IF im.v3_Avom.onStatus=statusDualInput.status_on THEN
	narabotka_izm:=DT_TO_UDINT( timer.CDT);
	timer.EN:=TRUE;
ELSE
	timer.EN:=FALSE;
END_IF
narabotka_hour (clk:=(narabotka_izm >=3600));
IF	narabotka_hour.Q THEN
	narabotka:=narabotka+1;
	timer.EN:=FALSE;
	narabotka_izm:=0;
END_IF
timer();

saveTimer(IN:=true);
IF saveTimer.Q THEN
	SaveToFile();
	saveTimer(IN:=FALSE);
END_IF*)

METHOD PROTECTED readPersistent
VAR_INPUT
END_VAR

narabotka:=STRING_TO_UDINT(readValue());
narabotka_izm:=STRING_TO_UDINT(readValue());
END_METHOD

METHOD PROTECTED writePersistent
VAR_INPUT
END_VAR

writeValue(value:= UDINT_TO_STRING(narabotka),'Наработка');
writeValue(value:= UDINT_TO_STRING(narabotka_izm),'Наработка_izm');
END_METHOD

END_FUNCTION_BLOCK

// K2/std12k5/Natabotka/Avom3
	{attribute 'symbol' := 'none'}
FUNCTION_BLOCK Avom3 EXTENDS Vent
VAR_INPUT
END_VAR
VAR_OUTPUT
		{attribute 'symbol' := 'read'}
	narabotka:UDINT;
	narabotka_:ExtNarabotka (table:=ADR (objectTable)):=(saveInterval:=T#1H);
END_VAR
VAR
	(*timer:RTC;	
	saveTimer:TON:=(PT:=T#600S);
	Narabotka_hour:R_TRIG;
	AvomStartted:R_TRIG;
	narabotka_Izm:UDINT;*)
END_VAR

SUPER^();
narabotka_.started:=onstatus=statusDualInput.STATUS_ON;
narabotka:=(narabotka_.narabotka/3600);
(*

AvomStartted(CLK:=im.v3_Avom.onStatus=statusDualInput.status_on);

	timer.PDT:=UDINT_TO_DT(narabotka_izm);

IF im.v3_Avom.onStatus=statusDualInput.status_on THEN
	narabotka_izm:=DT_TO_UDINT( timer.CDT);
	timer.EN:=TRUE;
ELSE
	timer.EN:=FALSE;
END_IF
narabotka_hour (clk:=(narabotka_izm >=3600));
IF	narabotka_hour.Q THEN
	narabotka:=narabotka+1;
	timer.EN:=FALSE;
	narabotka_izm:=0;
END_IF
timer();

saveTimer(IN:=true);
IF saveTimer.Q THEN
	SaveToFile();
	saveTimer(IN:=FALSE);
END_IF*)

METHOD PROTECTED readPersistent
VAR_INPUT
END_VAR

narabotka:=STRING_TO_UDINT(readValue());
narabotka_izm:=STRING_TO_UDINT(readValue());
END_METHOD

METHOD PROTECTED writePersistent
VAR_INPUT
END_VAR

writeValue(value:= UDINT_TO_STRING(narabotka),'Наработка');
writeValue(value:= UDINT_TO_STRING(narabotka_izm),'Наработка_izm');
END_METHOD

END_FUNCTION_BLOCK

// K1/std12k5/Narabotka/Avom4
	{attribute 'symbol' := 'none'}
FUNCTION_BLOCK Avom4 EXTENDS Vent
VAR_INPUT
END_VAR
VAR_OUTPUT
		{attribute 'symbol' := 'read'}
	narabotka:UDINT;
	narabotka_:ExtNarabotka (table:=ADR (objectTable)):=(saveInterval:=T#1H);
END_VAR
VAR
	(*timer:RTC;	
	saveTimer:TON:=(PT:=T#600S);
	Narabotka_hour:R_TRIG;
	AvomStartted:R_TRIG;
	narabotka_Izm:UDINT;*)
END_VAR

SUPER^();
narabotka_.started:=onstatus=statusDualInput.STATUS_ON;
narabotka:=(narabotka_.narabotka/3600);
(*
AvomStartted(CLK:=im.v4_Avom.onStatus=statusDualInput.status_on);

	timer.PDT:=UDINT_TO_DT(narabotka_izm);

IF im.v4_Avom.onStatus=statusDualInput.status_on THEN
	narabotka_izm:=DT_TO_UDINT( timer.CDT);
	timer.EN:=TRUE;
ELSE
	timer.EN:=FALSE;
END_IF
narabotka_hour (clk:=(narabotka_izm >=3600));
IF	narabotka_hour.Q THEN
	narabotka:=narabotka+1;
	timer.EN:=FALSE;
	narabotka_izm:=0;
END_IF
timer();

saveTimer(IN:=true);
IF saveTimer.Q THEN
	SaveToFile();
	saveTimer(IN:=FALSE);
END_IF*)

METHOD PROTECTED readPersistent
VAR_INPUT
END_VAR

narabotka:=STRING_TO_UDINT(readValue());
narabotka_izm:=STRING_TO_UDINT(readValue());
END_METHOD

METHOD PROTECTED writePersistent
VAR_INPUT
END_VAR

writeValue(value:= UDINT_TO_STRING(narabotka),'Наработка');
writeValue(value:= UDINT_TO_STRING(narabotka_izm),'Наработка_izm');
END_METHOD

END_FUNCTION_BLOCK

// K2/std12k5/Natabotka/Avom4
	{attribute 'symbol' := 'none'}
FUNCTION_BLOCK Avom4 EXTENDS Vent
VAR_INPUT
END_VAR
VAR_OUTPUT
		{attribute 'symbol' := 'read'}
	narabotka:UDINT;
	narabotka_:ExtNarabotka (table:=ADR (objectTable)):=(saveInterval:=T#1H);
END_VAR
VAR
(*	timer:RTC;	
	saveTimer:TON:=(PT:=T#600S);
	Narabotka_hour:R_TRIG;
	AvomStartted:R_TRIG;
	narabotka_Izm:UDINT;*)
END_VAR

SUPER^();
narabotka_.started:=onstatus=statusDualInput.STATUS_ON;
narabotka:=(narabotka_.narabotka/3600);

(*
AvomStartted(CLK:=im.v4_Avom.onStatus=statusDualInput.status_on);

	timer.PDT:=UDINT_TO_DT(narabotka_izm);

IF im.v4_Avom.onStatus=statusDualInput.status_on THEN
	narabotka_izm:=DT_TO_UDINT( timer.CDT);
	timer.EN:=TRUE;
ELSE
	timer.EN:=FALSE;
END_IF
narabotka_hour (clk:=(narabotka_izm >=3600));
IF	narabotka_hour.Q THEN
	narabotka:=narabotka+1;
	timer.EN:=FALSE;
	narabotka_izm:=0;
END_IF
timer();

saveTimer(IN:=true);
IF saveTimer.Q THEN
	SaveToFile();
	saveTimer(IN:=FALSE);
END_IF*)

METHOD PROTECTED readPersistent
VAR_INPUT
END_VAR

narabotka:=STRING_TO_UDINT(readValue());
narabotka_izm:=STRING_TO_UDINT(readValue());
END_METHOD

METHOD PROTECTED writePersistent
VAR_INPUT
END_VAR

writeValue(value:= UDINT_TO_STRING(narabotka),'Наработка');
writeValue(value:= UDINT_TO_STRING(narabotka_izm),'Наработка_izm');
END_METHOD

END_FUNCTION_BLOCK

// K1/std12k5/Ystavki/Delta_Vykl_AVOM1
	{attribute 'symbol' := 'none'}
FUNCTION_BLOCK Delta_Vykl_AVOM1 EXTENDS Baseobject
VAR_INPUT
	{attribute 'symbol' := 'readwright'}
	Yst_izm:UINT;
END_VAR
VAR_OUTPUT
	{attribute 'symbol' := 'read'}
	Yst_T1:UINT;
	
END_VAR
VAR
	Yst_Izm_trig:R_TRIG;
	Yst_First_izm:R_TRIG;
	flag:bool;
END_VAR

SUPER^();
Yst_Izm_trig(clk:=((Yst_izm <> Yst_T1) AND (Yst_izm >0) AND (Yst_izm <= 10)));
IF 	Yst_Izm_trig.Q THEN
	Yst_T1 := Yst_izm;
	SaveToFile();
END_IF	
Yst_First_izm(clk:=((Yst_izm = 0) AND (Yst_T1 = 0) AND flag));
IF	(Yst_izm = 0) AND (Yst_T1 = 0) AND flag THEN
	Yst_T1 := 1;
	Yst_izm := Yst_T1;
	SaveToFile();
END_IF;

flag:=true;

METHOD PROTECTED readPersistent
VAR_INPUT
END_VAR
Yst_izm:=STRING_TO_uint(readValue());
END_METHOD

METHOD PROTECTED writePersistent
VAR_INPUT
END_VAR
writeValue(value:= uint_TO_STRING(Yst_T1),'Наработка');
END_METHOD

END_FUNCTION_BLOCK

// K2/std12k5/Ystavki/Delta_Vykl_AVOM1
	{attribute 'symbol' := 'none'}
FUNCTION_BLOCK Delta_Vykl_AVOM1 EXTENDS Baseobject
VAR_INPUT
	{attribute 'symbol' := 'readwright'}
	Yst_izm:UINT;
END_VAR
VAR_OUTPUT
	{attribute 'symbol' := 'read'}
	Yst_T1:UINT;
	
END_VAR
VAR
	Yst_Izm_trig:R_TRIG;
	Yst_First_izm:R_TRIG;
	flag:bool;
END_VAR

SUPER^();
Yst_Izm_trig(clk:=((Yst_izm <> Yst_T1) AND (Yst_izm >0) AND (Yst_izm <= 10)));
IF 	Yst_Izm_trig.Q THEN
	Yst_T1 := Yst_izm;
	SaveToFile();
END_IF	
Yst_First_izm(clk:=((Yst_izm = 0) AND (Yst_T1 = 0) AND flag));
IF	(Yst_izm = 0) AND (Yst_T1 = 0) AND flag THEN
	Yst_T1 := 1;
	Yst_izm := Yst_T1;
	SaveToFile();
END_IF;

flag:=true;

METHOD PROTECTED readPersistent
VAR_INPUT
END_VAR
Yst_izm:=STRING_TO_uint(readValue());
END_METHOD

METHOD PROTECTED writePersistent
VAR_INPUT
END_VAR
writeValue(value:= uint_TO_STRING(Yst_T1),'Наработка');
END_METHOD

END_FUNCTION_BLOCK

// K1/std12k5/Ystavki/Delta_Vykl_AVOM2
	{attribute 'symbol' := 'none'}
FUNCTION_BLOCK Delta_Vykl_AVOM2 EXTENDS Baseobject
VAR_INPUT
	{attribute 'symbol' := 'readwright'}
	Yst_izm:UINT;
END_VAR
VAR_OUTPUT
	{attribute 'symbol' := 'read'}
	Yst_T2:UINT;
	
END_VAR
VAR
	Yst_Izm_trig:R_TRIG;
	Yst_First_izm:R_TRIG;
	flag:bool;
END_VAR

SUPER^();
Yst_Izm_trig(clk:=((Yst_izm <> Yst_T2) AND (Yst_izm > 0) AND (Yst_izm <=10)));
IF 	Yst_Izm_trig.Q THEN
	Yst_T2 := Yst_izm;
	SaveToFile();
END_IF	
Yst_First_izm(clk:=((Yst_izm = 0) AND (Yst_T2 = 0) AND flag));
IF	Yst_First_izm.Q	THEN
	Yst_T2 := 1;
	Yst_izm := Yst_T2;
	SaveToFile();
END_IF;
flag:=TRUE;

METHOD PROTECTED readPersistent
VAR_INPUT
END_VAR
Yst_izm:=STRING_TO_uint(readValue());
END_METHOD

METHOD PROTECTED writePersistent
VAR_INPUT
END_VAR
writeValue(value:= uint_TO_STRING(Yst_T2),'Наработка');
END_METHOD

END_FUNCTION_BLOCK

// K2/std12k5/Ystavki/Delta_Vykl_AVOM2
	{attribute 'symbol' := 'none'}
FUNCTION_BLOCK Delta_Vykl_AVOM2 EXTENDS Baseobject
VAR_INPUT
	{attribute 'symbol' := 'readwright'}
	Yst_izm:UINT;
END_VAR
VAR_OUTPUT
	{attribute 'symbol' := 'read'}
	Yst_T2:UINT;
	
END_VAR
VAR
	Yst_Izm_trig:R_TRIG;
	Yst_First_izm:R_TRIG;
	flag:bool;
END_VAR

SUPER^();
Yst_Izm_trig(clk:=((Yst_izm <> Yst_T2) AND (Yst_izm > 0) AND (Yst_izm <=10)));
IF 	Yst_Izm_trig.Q THEN
	Yst_T2 := Yst_izm;
	SaveToFile();
END_IF	
Yst_First_izm(clk:=((Yst_izm = 0) AND (Yst_T2 = 0) AND flag));
IF	Yst_First_izm.Q	THEN
	Yst_T2 := 1;
	Yst_izm := Yst_T2;
	SaveToFile();
END_IF;
flag:=TRUE;

METHOD PROTECTED readPersistent
VAR_INPUT
END_VAR
Yst_izm:=STRING_TO_uint(readValue());
END_METHOD

METHOD PROTECTED writePersistent
VAR_INPUT
END_VAR
writeValue(value:= uint_TO_STRING(Yst_T2),'Наработка');
END_METHOD

END_FUNCTION_BLOCK

// K1/std12k5/Ystavki/Delta_Vykl_AVOM3
	{attribute 'symbol' := 'none'}
FUNCTION_BLOCK Delta_Vykl_AVOM3 EXTENDS Baseobject
VAR_INPUT
	{attribute 'symbol' := 'readwright'}
	Yst_izm:UINT;
END_VAR
VAR_OUTPUT
	{attribute 'symbol' := 'read'}
	Yst_T3:UINT;
	
END_VAR
VAR
	flag:BOOL;
	Yst_Izm_trig:R_TRIG;
	Yst_First_izm:R_TRIG;
END_VAR

SUPER^();
Yst_Izm_trig(clk:=((Yst_izm <> Yst_T3) AND (Yst_izm >0) AND (Yst_izm <= 10)));
IF 	Yst_Izm_trig.Q THEN
	Yst_T3 := Yst_izm;
	SaveToFile();
END_IF	
Yst_First_izm(clk:=((Yst_izm = 0) AND (Yst_T3 = 0) AND flag));
IF	Yst_First_izm.Q THEN
	Yst_T3 := 1;
	Yst_izm := Yst_T3;
	SaveToFile();
END_IF;
flag:=true;

METHOD PROTECTED readPersistent
VAR_INPUT
END_VAR

Yst_izm:=STRING_TO_uint(readValue());
END_METHOD

METHOD PROTECTED writePersistent
VAR_INPUT
END_VAR

writeValue(value:= uint_TO_STRING(Yst_T3),'Наработка');
END_METHOD

END_FUNCTION_BLOCK

// K2/std12k5/Ystavki/Delta_Vykl_AVOM3
	{attribute 'symbol' := 'none'}
FUNCTION_BLOCK Delta_Vykl_AVOM3 EXTENDS Baseobject
VAR_INPUT
	{attribute 'symbol' := 'readwright'}
	Yst_izm:UINT;
END_VAR
VAR_OUTPUT
	{attribute 'symbol' := 'read'}
	Yst_T3:UINT;
	
END_VAR
VAR
	flag:BOOL;
	Yst_Izm_trig:R_TRIG;
	Yst_First_izm:R_TRIG;
END_VAR

SUPER^();
Yst_Izm_trig(clk:=((Yst_izm <> Yst_T3) AND (Yst_izm >0) AND (Yst_izm <= 10)));
IF 	Yst_Izm_trig.Q THEN
	Yst_T3 := Yst_izm;
	SaveToFile();
END_IF	
Yst_First_izm(clk:=((Yst_izm = 0) AND (Yst_T3 = 0) AND flag));
IF	Yst_First_izm.Q THEN
	Yst_T3 := 1;
	Yst_izm := Yst_T3;
	SaveToFile();
END_IF;
flag:=true;

METHOD PROTECTED readPersistent
VAR_INPUT
END_VAR

Yst_izm:=STRING_TO_uint(readValue());
END_METHOD

METHOD PROTECTED writePersistent
VAR_INPUT
END_VAR

writeValue(value:= uint_TO_STRING(Yst_T3),'Наработка');
END_METHOD

END_FUNCTION_BLOCK

// K1/std12k5/Ystavki/Delta_Vykl_AVOM4
	{attribute 'symbol' := 'none'}
FUNCTION_BLOCK Delta_Vykl_AVOM4 EXTENDS Baseobject
VAR_INPUT
	{attribute 'symbol' := 'readwright'}
	Yst_izm:UINT;
END_VAR
VAR_OUTPUT
	{attribute 'symbol' := 'read'}
	Yst_T4:UINT;
	
END_VAR
VAR
	flag:BOOL;
	Yst_Izm_trig:R_TRIG;
	Yst_First_izm:R_TRIG;
END_VAR

SUPER^();
Yst_Izm_trig(clk:=((Yst_izm <> Yst_T4) AND (Yst_izm > 0) AND (Yst_izm <= 10)));
IF 	Yst_Izm_trig.Q THEN
	Yst_T4 := Yst_izm;
	SaveToFile();
END_IF	
Yst_First_izm(clk:=((Yst_izm = 0) AND (Yst_T4 = 0) AND flag));
IF	Yst_First_izm.Q THEN
	Yst_T4 := 1;
	Yst_izm := Yst_T4;
	SaveToFile();
END_IF;

flag:=TRUE;

METHOD PROTECTED readPersistent
VAR_INPUT
END_VAR

Yst_izm:=STRING_TO_uint(readValue());
END_METHOD

METHOD PROTECTED writePersistent
VAR_INPUT
END_VAR

writeValue(value:= uint_TO_STRING(Yst_T4),'Наработка');
END_METHOD

END_FUNCTION_BLOCK

// K2/std12k5/Ystavki/Delta_Vykl_AVOM4
	{attribute 'symbol' := 'none'}
FUNCTION_BLOCK Delta_Vykl_AVOM4 EXTENDS Baseobject
VAR_INPUT
	{attribute 'symbol' := 'readwright'}
	Yst_izm:UINT;
END_VAR
VAR_OUTPUT
	{attribute 'symbol' := 'read'}
	Yst_T4:UINT;
	
END_VAR
VAR
	flag:BOOL;
	Yst_Izm_trig:R_TRIG;
	Yst_First_izm:R_TRIG;
END_VAR

SUPER^();
Yst_Izm_trig(clk:=((Yst_izm <> Yst_T4) AND (Yst_izm > 0) AND (Yst_izm <= 10)));
IF 	Yst_Izm_trig.Q THEN
	Yst_T4 := Yst_izm;
	SaveToFile();
END_IF	
Yst_First_izm(clk:=((Yst_izm = 0) AND (Yst_T4 = 0) AND flag));
IF	Yst_First_izm.Q THEN
	Yst_T4 := 1;
	Yst_izm := Yst_T4;
	SaveToFile();
END_IF;

flag:=TRUE;

METHOD PROTECTED readPersistent
VAR_INPUT
END_VAR

Yst_izm:=STRING_TO_uint(readValue());
END_METHOD

METHOD PROTECTED writePersistent
VAR_INPUT
END_VAR

writeValue(value:= uint_TO_STRING(Yst_T4),'Наработка');
END_METHOD

END_FUNCTION_BLOCK

// K1/std12k5/Narabotka/EO
	{attribute 'symbol' := 'none'}
FUNCTION_BLOCK EO EXTENDS BaseIM
VAR_INPUT
END_VAR
VAR_OUTPUT
	
		{attribute 'symbol' := 'read'}
	narabotka:UDINT;
END_VAR
VAR
	Work_End:F_TRIG;
	flag:bool;
	AvomStartted:R_TRIG;
END_VAR

SUPER^();
Work_END (CLK:=(algmanager.mode=modegpa.MODE_WORK_K OR algmanager.mode=modegpa.MODE_WORK_M));
IF Work_END.Q THEN
	flag:=TRUE;
END_IF
AvomStartted(CLK:=(algmanager.mode=modegpa.MODE_EO) AND flag);
IF AvomStartted.Q THEN
	narabotka:= narabotka + 1;
	SaveToFile();
	flag:=false;
END_IF

METHOD PROTECTED readPersistent
VAR_INPUT
END_VAR

narabotka:=STRING_TO_UDINT(readValue());
END_METHOD

METHOD PROTECTED writePersistent
VAR_INPUT
END_VAR

writeValue(value:= UDINT_TO_STRING(narabotka),'Наработка');
END_METHOD

END_FUNCTION_BLOCK

// K2/std12k5/Natabotka/EO
	{attribute 'symbol' := 'none'}
FUNCTION_BLOCK EO EXTENDS BaseIM
VAR_INPUT
END_VAR
VAR_OUTPUT
	
		{attribute 'symbol' := 'read'}
	narabotka:UDINT;
END_VAR
VAR
	Work_End:F_TRIG;
	flag:bool;
	AvomStartted:R_TRIG;
END_VAR

SUPER^();
Work_END (CLK:=(algmanager.mode=modegpa.MODE_WORK_K OR algmanager.mode=modegpa.MODE_WORK_M));
IF Work_END.Q THEN
	flag:=TRUE;
END_IF
AvomStartted(CLK:=(algmanager.mode=modegpa.MODE_EO) AND flag);
IF AvomStartted.Q THEN
	narabotka:= narabotka + 1;
	SaveToFile();
	flag:=false;
END_IF

METHOD PROTECTED readPersistent
VAR_INPUT
END_VAR

narabotka:=STRING_TO_UDINT(readValue());
END_METHOD

METHOD PROTECTED writePersistent
VAR_INPUT
END_VAR

writeValue(value:= UDINT_TO_STRING(narabotka),'Наработка');
END_METHOD

END_FUNCTION_BLOCK

// K1/std12k5/Narabotka/nu1
	{attribute 'symbol' := 'none'}
FUNCTION_BLOCK nu1 EXTENDS nasos
VAR_INPUT
END_VAR
VAR_OUTPUT
	
		{attribute 'symbol' := 'read'}
	narabotka:UDINT;
	narabotka_:ExtNarabotka (table:=ADR (objectTable)):=(saveInterval:=T#1H);
END_VAR
VAR
	(*	timer:RTC;	
	saveTimer:TON:=(PT:=T#600S);
	Narabotka_hour:R_TRIG;
	AvomStartted:R_TRIG;
	narabotka_Izm:UDINT;*)
END_VAR

SUPER^();
narabotka_.started:=im.nu.nu1.onStatus=statusDualInput.STATUS_ON;
narabotka:=(narabotka_.narabotka/3600);
(*
AvomStartted(CLK:=im.nu.nu1.onStatus=statusDualInput.status_on);

	timer.PDT:=UDINT_TO_DT(narabotka_izm);

IF im.nu.nu1.onStatus=statusDualInput.status_on THEN
	narabotka_izm:=DT_TO_UDINT( timer.CDT);
	timer.EN:=TRUE;
ELSE
	timer.EN:=FALSE;
END_IF
narabotka_hour (clk:=(narabotka_izm >=3600));
IF	narabotka_hour.Q THEN
	narabotka:=narabotka+1;
	timer.EN:=FALSE;
	narabotka_izm:=0;
END_IF
timer();

saveTimer(IN:=true);
IF saveTimer.Q THEN
	SaveToFile();
	saveTimer(IN:=FALSE);
END_IF*)

METHOD PROTECTED readPersistent
VAR_INPUT
END_VAR

narabotka:=STRING_TO_UDINT(readValue());
narabotka_izm:=STRING_TO_UDINT(readValue());
END_METHOD

METHOD PROTECTED writePersistent
VAR_INPUT
END_VAR

writeValue(value:= UDINT_TO_STRING(narabotka),'Наработка');
writeValue(value:= UDINT_TO_STRING(narabotka_izm),'Наработка_izm');
END_METHOD

END_FUNCTION_BLOCK

// K2/std12k5/Natabotka/nu1
	{attribute 'symbol' := 'none'}
FUNCTION_BLOCK nu1 EXTENDS nasos
VAR_INPUT
END_VAR
VAR_OUTPUT
	
		{attribute 'symbol' := 'read'}
	narabotka:UDINT;
	narabotka_:ExtNarabotka (table:=ADR (objectTable)):=(saveInterval:=T#1H);
END_VAR
VAR
	(*	timer:RTC;	
	saveTimer:TON:=(PT:=T#600S);
	Narabotka_hour:R_TRIG;
	AvomStartted:R_TRIG;
	narabotka_Izm:UDINT;*)
END_VAR

SUPER^();
narabotka_.started:=im.nu.nu1.onStatus=statusDualInput.STATUS_ON;
narabotka:=(narabotka_.narabotka/3600);
(*
AvomStartted(CLK:=im.nu.nu1.onStatus=statusDualInput.status_on);

	timer.PDT:=UDINT_TO_DT(narabotka_izm);

IF im.nu.nu1.onStatus=statusDualInput.status_on THEN
	narabotka_izm:=DT_TO_UDINT( timer.CDT);
	timer.EN:=TRUE;
ELSE
	timer.EN:=FALSE;
END_IF
narabotka_hour (clk:=(narabotka_izm >=3600));
IF	narabotka_hour.Q THEN
	narabotka:=narabotka+1;
	timer.EN:=FALSE;
	narabotka_izm:=0;
END_IF
timer();

saveTimer(IN:=true);
IF saveTimer.Q THEN
	SaveToFile();
	saveTimer(IN:=FALSE);
END_IF*)

METHOD PROTECTED readPersistent
VAR_INPUT
END_VAR

narabotka:=STRING_TO_UDINT(readValue());
narabotka_izm:=STRING_TO_UDINT(readValue());
END_METHOD

METHOD PROTECTED writePersistent
VAR_INPUT
END_VAR

writeValue(value:= UDINT_TO_STRING(narabotka),'Наработка');
writeValue(value:= UDINT_TO_STRING(narabotka_izm),'Наработка_izm');
END_METHOD

END_FUNCTION_BLOCK

// lowLevel_ecl/im/ventvs/Nasos
	{attribute 'symbol' := 'none'}
FUNCTION_BLOCK Nasos EXTENDS Ventvs
VAR_INPUT
END_VAR
VAR_OUTPUT
END_VAR
VAR
END_VAR

SUPER^();

END_FUNCTION_BLOCK

// K1/std12k5/Narabotka/nu2
	{attribute 'symbol' := 'none'}
FUNCTION_BLOCK nu2 EXTENDS Nasos
VAR_INPUT
END_VAR
VAR_OUTPUT
	
		{attribute 'symbol' := 'read'}
	narabotka:UDINT;
	narabotka_:ExtNarabotka (table:=ADR (objectTable)):=(saveInterval:=T#1H);
END_VAR
VAR
(*	timer:RTC;	
	saveTimer:TON:=(PT:=T#600S);
	Narabotka_hour:R_TRIG;
	AvomStartted:R_TRIG;
	narabotka_Izm:UDINT;*)
END_VAR

SUPER^();
narabotka_.started:=im.nu.nu2.onStatus=statusDualInput.STATUS_ON;
narabotka:=(narabotka_.narabotka/3600);
(*
AvomStartted(CLK:=im.nu.nu2.onStatus=statusDualInput.status_on);

	timer.PDT:=UDINT_TO_DT(narabotka_izm);

IF im.nu.nu2.onStatus=statusDualInput.status_on THEN
	narabotka_izm:=DT_TO_UDINT( timer.CDT);
	timer.EN:=TRUE;
ELSE
	timer.EN:=FALSE;
END_IF
narabotka_hour (clk:=(narabotka_izm >=3600));
IF	narabotka_hour.Q THEN
	narabotka:=narabotka+1;
	timer.EN:=FALSE;
	narabotka_izm:=0;
END_IF
timer();

saveTimer(IN:=true);
IF saveTimer.Q THEN
	SaveToFile();
	saveTimer(IN:=FALSE);
END_IF*)

METHOD PROTECTED readPersistent
VAR_INPUT
END_VAR

narabotka:=STRING_TO_UDINT(readValue());
narabotka_izm:=STRING_TO_UDINT(readValue());
END_METHOD

METHOD PROTECTED writePersistent
VAR_INPUT
END_VAR

writeValue(value:= UDINT_TO_STRING(narabotka),'Наработка');
writeValue(value:= UDINT_TO_STRING(narabotka_izm),'Наработка_izm');
END_METHOD

END_FUNCTION_BLOCK

// K2/std12k5/Natabotka/nu2
	{attribute 'symbol' := 'none'}
FUNCTION_BLOCK nu2 EXTENDS Nasos
VAR_INPUT
END_VAR
VAR_OUTPUT
	
		{attribute 'symbol' := 'read'}
	narabotka:UDINT;
	narabotka_:ExtNarabotka (table:=ADR (objectTable)):=(saveInterval:=T#1H);
END_VAR
VAR
(*	timer:RTC;	
	saveTimer:TON:=(PT:=T#600S);
	Narabotka_hour:R_TRIG;
	AvomStartted:R_TRIG;
	narabotka_Izm:UDINT;*)
END_VAR

SUPER^();
narabotka_.started:=im.nu.nu2.onStatus=statusDualInput.STATUS_ON;
narabotka:=(narabotka_.narabotka/3600);
(*
AvomStartted(CLK:=im.nu.nu2.onStatus=statusDualInput.status_on);

	timer.PDT:=UDINT_TO_DT(narabotka_izm);

IF im.nu.nu2.onStatus=statusDualInput.status_on THEN
	narabotka_izm:=DT_TO_UDINT( timer.CDT);
	timer.EN:=TRUE;
ELSE
	timer.EN:=FALSE;
END_IF
narabotka_hour (clk:=(narabotka_izm >=3600));
IF	narabotka_hour.Q THEN
	narabotka:=narabotka+1;
	timer.EN:=FALSE;
	narabotka_izm:=0;
END_IF
timer();

saveTimer(IN:=true);
IF saveTimer.Q THEN
	SaveToFile();
	saveTimer(IN:=FALSE);
END_IF*)

METHOD PROTECTED readPersistent
VAR_INPUT
END_VAR

narabotka:=STRING_TO_UDINT(readValue());
narabotka_izm:=STRING_TO_UDINT(readValue());
END_METHOD

METHOD PROTECTED writePersistent
VAR_INPUT
END_VAR

writeValue(value:= UDINT_TO_STRING(narabotka),'Наработка');
writeValue(value:= UDINT_TO_STRING(narabotka_izm),'Наработка_izm');
END_METHOD

END_FUNCTION_BLOCK

// K1/std12k5/Narabotka/pns_
	{attribute 'symbol' := 'none'}
FUNCTION_BLOCK pns_ EXTENDS nasos
VAR_INPUT
END_VAR
VAR_OUTPUT
	
		{attribute 'symbol' := 'read'}
	narabotka:UDINT;
	narabotka_:ExtNarabotka (table:=ADR (objectTable)):=(saveInterval:=T#1H);
END_VAR
VAR
(*	timer:RTC;	
	saveTimer:TON:=(PT:=T#600S);
	Narabotka_hour:R_TRIG;
	AvomStartted:R_TRIG;
	narabotka_Izm:UDINT;*)
END_VAR

SUPER^();
narabotka_.started:=onStatus=statusDualInput.STATUS_ON;
narabotka:=(narabotka_.narabotka/3600);
(*
AvomStartted(CLK:=im.PNS.onStatus=statusDualInput.status_on);

	timer.PDT:=UDINT_TO_DT(narabotka_izm);

IF im.PNS.onStatus=statusDualInput.status_on THEN
	narabotka_izm:=DT_TO_UDINT( timer.CDT);
	timer.EN:=TRUE;
ELSE
	timer.EN:=FALSE;
END_IF
narabotka_hour (clk:=(narabotka_izm >=3600));
IF	narabotka_hour.Q THEN
	narabotka:=narabotka+1;
	timer.EN:=FALSE;
	narabotka_izm:=0;
END_IF
timer();

saveTimer(IN:=true);
IF saveTimer.Q THEN
	SaveToFile();
	saveTimer(IN:=FALSE);
END_IF*)

METHOD PROTECTED readPersistent
VAR_INPUT
END_VAR

narabotka:=STRING_TO_UDINT(readValue());
narabotka_izm:=STRING_TO_UDINT(readValue());
END_METHOD

METHOD PROTECTED writePersistent
VAR_INPUT
END_VAR

writeValue(value:= UDINT_TO_STRING(narabotka),'Наработка');
writeValue(value:= UDINT_TO_STRING(narabotka_izm),'Наработка_izm');
END_METHOD

END_FUNCTION_BLOCK

// K2/std12k5/Natabotka/pns_
	{attribute 'symbol' := 'none'}
FUNCTION_BLOCK pns_ EXTENDS nasos
VAR_INPUT
END_VAR
VAR_OUTPUT
	
		{attribute 'symbol' := 'read'}
	narabotka:UDINT;
		narabotka_:ExtNarabotka (table:=ADR (objectTable)):=(saveInterval:=T#1H);
END_VAR
VAR
	(*timer:RTC;	
	saveTimer:TON:=(PT:=T#600S);
	Narabotka_hour:R_TRIG;
	AvomStartted:R_TRIG;
	narabotka_Izm:UDINT;*)
END_VAR

SUPER^();
narabotka_.started:=onStatus=statusDualInput.STATUS_ON;
narabotka:=(narabotka_.narabotka/3600);
(*
AvomStartted(CLK:=im.PNS.onStatus=statusDualInput.status_on);

	timer.PDT:=UDINT_TO_DT(narabotka_izm);

IF im.PNS.onStatus=statusDualInput.status_on THEN
	narabotka_izm:=DT_TO_UDINT( timer.CDT);
	timer.EN:=TRUE;
ELSE
	timer.EN:=FALSE;
END_IF
narabotka_hour (clk:=(narabotka_izm >=3600));
IF	narabotka_hour.Q THEN
	narabotka:=narabotka+1;
	timer.EN:=FALSE;
	narabotka_izm:=0;
END_IF
timer();

saveTimer(IN:=true);
IF saveTimer.Q THEN
	SaveToFile();
	saveTimer(IN:=FALSE);
END_IF*)

METHOD PROTECTED readPersistent
VAR_INPUT
END_VAR

narabotka:=STRING_TO_UDINT(readValue());
narabotka_izm:=STRING_TO_UDINT(readValue());
END_METHOD

METHOD PROTECTED writePersistent
VAR_INPUT
END_VAR

writeValue(value:= UDINT_TO_STRING(narabotka),'Наработка');
writeValue(value:= UDINT_TO_STRING(narabotka_izm),'Наработка_izm');
END_METHOD

END_FUNCTION_BLOCK

// K1/std12k5/Narabotka/Pusk
	{attribute 'symbol' := 'none'}
FUNCTION_BLOCK Pusk EXTENDS BaseIM
VAR_INPUT
END_VAR
VAR_OUTPUT
	
		{attribute 'symbol' := 'read'}
	narabotka:UDINT;
END_VAR
VAR
	
	
	AvomStartted:R_TRIG;
END_VAR

SUPER^();

AvomStartted(CLK:=(algmanager.mode=modegpa.MODE_WORK_K) OR (algmanager.mode=modegpa.MODE_WORK_M));
IF AvomStartted.Q THEN
	narabotka:= narabotka + 1;
	SaveToFile();
END_IF

METHOD PROTECTED readPersistent
VAR_INPUT
END_VAR

narabotka:=STRING_TO_UDINT(readValue());
END_METHOD

METHOD PROTECTED writePersistent
VAR_INPUT
END_VAR

writeValue(value:= UDINT_TO_STRING(narabotka),'Наработка');
END_METHOD

END_FUNCTION_BLOCK

// K2/std12k5/Natabotka/Pusk
	{attribute 'symbol' := 'none'}
FUNCTION_BLOCK Pusk EXTENDS BaseIM
VAR_INPUT
END_VAR
VAR_OUTPUT
	
		{attribute 'symbol' := 'read'}
	narabotka:UDINT;
END_VAR
VAR
	
	
	AvomStartted:R_TRIG;
END_VAR

SUPER^();

AvomStartted(CLK:=(algmanager.mode=modegpa.MODE_WORK_K) OR (algmanager.mode=modegpa.MODE_WORK_M));
IF AvomStartted.Q THEN
	narabotka:= narabotka + 1;
	SaveToFile();
END_IF

METHOD PROTECTED readPersistent
VAR_INPUT
END_VAR

narabotka:=STRING_TO_UDINT(readValue());
END_METHOD

METHOD PROTECTED writePersistent
VAR_INPUT
END_VAR

writeValue(value:= UDINT_TO_STRING(narabotka),'Наработка');
END_METHOD

END_FUNCTION_BLOCK

// K1/std12k5/Ystavki/T1_AVOM
	{attribute 'symbol' := 'none'}
FUNCTION_BLOCK T1_AVOM EXTENDS Baseobject
VAR_INPUT
	{attribute 'symbol' := 'readwright'}
	Yst_izm:UINT;
END_VAR
VAR_OUTPUT
	{attribute 'symbol' := 'read'}
	Yst_T1:UINT;
	
END_VAR
VAR
	flag:BOOL;
	Yst_Izm_trig:R_TRIG;
	Yst_First_izm:R_TRIG;
END_VAR

SUPER^();
Yst_Izm_trig(clk:=((Yst_izm <> Yst_T1) 	AND (Yst_izm > 0) AND (Yst_izm < 100) AND (Yst_izm < Ystavki.Yst_AVOM_T2.Yst_T2)));
IF 	Yst_Izm_trig.Q THEN
	Yst_T1 := Yst_izm;
	SaveToFile();
END_IF	
Yst_First_izm(clk:=((Yst_izm = 0) AND (Yst_T1 = 0) AND flag));
IF	Yst_First_izm.Q  THEN
	Yst_T1 := 41;
	Yst_izm := Yst_T1;
	SaveToFile();
END_IF;

flag:=true;

METHOD PROTECTED readPersistent
VAR_INPUT
END_VAR

Yst_izm:=STRING_TO_uint(readValue());
END_METHOD

METHOD PROTECTED writePersistent
VAR_INPUT
END_VAR

writeValue(value:= uint_TO_STRING(Yst_T1),'Наработка');
END_METHOD

END_FUNCTION_BLOCK

// K2/std12k5/Ystavki/T1_AVOM
	{attribute 'symbol' := 'none'}
FUNCTION_BLOCK T1_AVOM EXTENDS Baseobject
VAR_INPUT
	{attribute 'symbol' := 'readwright'}
	Yst_izm:UINT;
END_VAR
VAR_OUTPUT
	{attribute 'symbol' := 'read'}
	Yst_T1:UINT;
	
END_VAR
VAR
	flag:BOOL;
	Yst_Izm_trig:R_TRIG;
	Yst_First_izm:R_TRIG;
END_VAR

SUPER^();
Yst_Izm_trig(clk:=((Yst_izm <> Yst_T1) 	AND (Yst_izm > 0) AND (Yst_izm < 100) AND (Yst_izm < Ystavki.Yst_AVOM_T2.Yst_T2)));
IF 	Yst_Izm_trig.Q THEN
	Yst_T1 := Yst_izm;
	SaveToFile();
END_IF	
Yst_First_izm(clk:=((Yst_izm = 0) AND (Yst_T1 = 0) AND flag));
IF	Yst_First_izm.Q  THEN
	Yst_T1 := 41;
	Yst_izm := Yst_T1;
	SaveToFile();
END_IF;

flag:=true;

METHOD PROTECTED readPersistent
VAR_INPUT
END_VAR

Yst_izm:=STRING_TO_uint(readValue());
END_METHOD

METHOD PROTECTED writePersistent
VAR_INPUT
END_VAR

writeValue(value:= uint_TO_STRING(Yst_T1),'Наработка');
END_METHOD

END_FUNCTION_BLOCK

// K1/std12k5/Ystavki/T2_AVOM
	{attribute 'symbol' := 'none'}
FUNCTION_BLOCK T2_AVOM EXTENDS Baseobject
VAR_INPUT
	{attribute 'symbol' := 'readwright'}
	Yst_izm:UINT;
END_VAR
VAR_OUTPUT
	{attribute 'symbol' := 'read'}
	Yst_T2:UINT;
	
END_VAR
VAR
	flag:BOOL;
	Yst_Izm_trig:R_TRIG;
	Yst_First_izm:R_TRIG;
END_VAR

SUPER^();
Yst_Izm_trig(clk:=((Yst_izm <> Yst_T2) 	AND (Yst_izm >0) AND (Yst_izm < 100) AND (Yst_izm > Ystavki.Yst_AVOM_T1.Yst_T1) AND (Yst_izm < Ystavki.Yst_AVOM_T3.Yst_T3)));
IF 	Yst_Izm_trig.Q THEN
	Yst_T2 := Yst_izm;
	SaveToFile();
END_IF	
Yst_First_izm(clk:=((Yst_izm = 0) AND (Yst_T2 = 0) AND flag ));
IF	Yst_First_izm.Q THEN
	Yst_T2 := 42;
	Yst_izm := Yst_T2;
	SaveToFile();
END_IF;



flag:=TRUE;

METHOD PROTECTED readPersistent
VAR_INPUT
END_VAR

Yst_izm:=STRING_TO_uint(readValue());
END_METHOD

METHOD PROTECTED writePersistent
VAR_INPUT
END_VAR

writeValue(value:= uint_TO_STRING(Yst_T2),'Наработка');
END_METHOD

END_FUNCTION_BLOCK

// K2/std12k5/Ystavki/T2_AVOM
	{attribute 'symbol' := 'none'}
FUNCTION_BLOCK T2_AVOM EXTENDS Baseobject
VAR_INPUT
	{attribute 'symbol' := 'readwright'}
	Yst_izm:UINT;
END_VAR
VAR_OUTPUT
	{attribute 'symbol' := 'read'}
	Yst_T2:UINT;
	
END_VAR
VAR
	flag:BOOL;
	Yst_Izm_trig:R_TRIG;
	Yst_First_izm:R_TRIG;
END_VAR

SUPER^();
Yst_Izm_trig(clk:=((Yst_izm <> Yst_T2) 	AND (Yst_izm >0) AND (Yst_izm < 100) AND (Yst_izm > Ystavki.Yst_AVOM_T1.Yst_T1) AND (Yst_izm < Ystavki.Yst_AVOM_T3.Yst_T3)));
IF 	Yst_Izm_trig.Q THEN
	Yst_T2 := Yst_izm;
	SaveToFile();
END_IF	
Yst_First_izm(clk:=((Yst_izm = 0) AND (Yst_T2 = 0) AND flag ));
IF	Yst_First_izm.Q THEN
	Yst_T2 := 42;
	Yst_izm := Yst_T2;
	SaveToFile();
END_IF;



flag:=TRUE;

METHOD PROTECTED readPersistent
VAR_INPUT
END_VAR

Yst_izm:=STRING_TO_uint(readValue());
END_METHOD

METHOD PROTECTED writePersistent
VAR_INPUT
END_VAR

writeValue(value:= uint_TO_STRING(Yst_T2),'Наработка');
END_METHOD

END_FUNCTION_BLOCK

// K1/std12k5/Ystavki/T3_AVOM
	{attribute 'symbol' := 'none'}
FUNCTION_BLOCK T3_AVOM EXTENDS Baseobject
VAR_INPUT
		
	
{attribute 'symbol' := 'readwright'}
	Yst_izm:UINT;
END_VAR
VAR_OUTPUT
	{attribute 'symbol' := 'read'}
	Yst_T3:UINT;
END_VAR
VAR
	flag:BOOL;
	Yst_Izm_trig:R_TRIG;
	Yst_First_izm:R_TRIG;
END_VAR

SUPER^();
Yst_Izm_trig(clk:=((Yst_izm <> Yst_T3) 	AND (Yst_izm >0) AND (Yst_izm < 100) AND (Yst_izm > ystavki.Yst_AVOM_T2.Yst_T2) AND (Yst_izm < ystavki.Yst_AVOM_T4.Yst_T4)));
IF 	Yst_Izm_trig.Q	THEN
	Yst_T3 := Yst_izm;
	SaveToFile();
END_IF	
Yst_First_izm(clk:=((Yst_izm = 0) AND (Yst_T3 = 0) AND flag));
IF	Yst_First_izm.Q THEN
	Yst_T3 := 43;
	Yst_izm := Yst_T3;
	SaveToFile();
END_IF;


flag:=TRUE;

METHOD PROTECTED readPersistent
VAR_INPUT
END_VAR

Yst_izm:=STRING_TO_uint(readValue());
END_METHOD

METHOD PROTECTED writePersistent
VAR_INPUT
END_VAR

writeValue(value:= uint_TO_STRING(Yst_T3),'Наработка');
END_METHOD

END_FUNCTION_BLOCK

// K2/std12k5/Ystavki/T3_AVOM
	{attribute 'symbol' := 'none'}
FUNCTION_BLOCK T3_AVOM EXTENDS Baseobject
VAR_INPUT
		
	
{attribute 'symbol' := 'readwright'}
	Yst_izm:UINT;
END_VAR
VAR_OUTPUT
	{attribute 'symbol' := 'read'}
	Yst_T3:UINT;
END_VAR
VAR
	flag:BOOL;
	Yst_Izm_trig:R_TRIG;
	Yst_First_izm:R_TRIG;
END_VAR

SUPER^();
Yst_Izm_trig(clk:=((Yst_izm <> Yst_T3) 	AND (Yst_izm >0) AND (Yst_izm < 100) AND (Yst_izm > ystavki.Yst_AVOM_T2.Yst_T2) AND (Yst_izm < ystavki.Yst_AVOM_T4.Yst_T4)));
IF 	Yst_Izm_trig.Q	THEN
	Yst_T3 := Yst_izm;
	SaveToFile();
END_IF	
Yst_First_izm(clk:=((Yst_izm = 0) AND (Yst_T3 = 0) AND flag));
IF	Yst_First_izm.Q THEN
	Yst_T3 := 43;
	Yst_izm := Yst_T3;
	SaveToFile();
END_IF;


flag:=TRUE;

METHOD PROTECTED readPersistent
VAR_INPUT
END_VAR

Yst_izm:=STRING_TO_uint(readValue());
END_METHOD

METHOD PROTECTED writePersistent
VAR_INPUT
END_VAR

writeValue(value:= uint_TO_STRING(Yst_T3),'Наработка');
END_METHOD

END_FUNCTION_BLOCK

// K1/std12k5/Ystavki/T4_AVOM
	{attribute 'symbol' := 'none'}
FUNCTION_BLOCK T4_AVOM EXTENDS Baseobject
VAR_INPUT
	{attribute 'symbol' := 'readwright'}
	Yst_izm:UINT;
END_VAR
VAR_OUTPUT
	{attribute 'symbol' := 'read'}
	Yst_T4:UINT;
	
END_VAR
VAR
	flag:BOOL;
	Yst_Izm_trig:R_TRIG;
	Yst_First_izm:R_TRIG;
END_VAR

SUPER^();
Yst_Izm_trig(clk:=((Yst_izm <> Yst_T4) 	AND (Yst_izm >0) AND (Yst_izm < 100) AND (Yst_izm > Ystavki.Yst_AVOM_T3.Yst_T3)));
IF 	Yst_Izm_trig.Q THEN
	Yst_T4 := Yst_izm;
	SaveToFile();
END_IF	
Yst_First_izm(clk:=((Yst_izm = 0) AND (Yst_T4 = 0) AND flag ));
IF	Yst_First_izm.Q THEN
	Yst_T4 := 44;
	Yst_izm := Yst_T4;
	SaveToFile();
END_IF;

flag:=TRUE;

METHOD PROTECTED readPersistent
VAR_INPUT
END_VAR

Yst_izm:=STRING_TO_uint(readValue());
END_METHOD

METHOD PROTECTED writePersistent
VAR_INPUT
END_VAR

writeValue(value:= uint_TO_STRING(Yst_T4),'Наработка');
END_METHOD

END_FUNCTION_BLOCK

// K2/std12k5/Ystavki/T4_AVOM
	{attribute 'symbol' := 'none'}
FUNCTION_BLOCK T4_AVOM EXTENDS Baseobject
VAR_INPUT
	{attribute 'symbol' := 'readwright'}
	Yst_izm:UINT;
END_VAR
VAR_OUTPUT
	{attribute 'symbol' := 'read'}
	Yst_T4:UINT;
	
END_VAR
VAR
	flag:BOOL;
	Yst_Izm_trig:R_TRIG;
	Yst_First_izm:R_TRIG;
END_VAR

SUPER^();
Yst_Izm_trig(clk:=((Yst_izm <> Yst_T4) 	AND (Yst_izm >0) AND (Yst_izm < 100) AND (Yst_izm > Ystavki.Yst_AVOM_T3.Yst_T3)));
IF 	Yst_Izm_trig.Q THEN
	Yst_T4 := Yst_izm;
	SaveToFile();
END_IF	
Yst_First_izm(clk:=((Yst_izm = 0) AND (Yst_T4 = 0) AND flag ));
IF	Yst_First_izm.Q THEN
	Yst_T4 := 44;
	Yst_izm := Yst_T4;
	SaveToFile();
END_IF;

flag:=TRUE;

METHOD PROTECTED readPersistent
VAR_INPUT
END_VAR

Yst_izm:=STRING_TO_uint(readValue());
END_METHOD

METHOD PROTECTED writePersistent
VAR_INPUT
END_VAR

writeValue(value:= uint_TO_STRING(Yst_T4),'Наработка');
END_METHOD

END_FUNCTION_BLOCK

// K1/std12k5/Ystavki/Tvkl_AVOM1
	{attribute 'symbol' := 'none'}
FUNCTION_BLOCK Tvkl_AVOM1 EXTENDS Baseobject
VAR_INPUT
	{attribute 'symbol' := 'readwright'}
	Yst_izm:UINT;
END_VAR
VAR_OUTPUT
	{attribute 'symbol' := 'read'}
	Yst_T1:UINT;
	
END_VAR
VAR
	flag:BOOL;
	Yst_Izm_trig:R_TRIG;
	Yst_First_izm:R_TRIG;
END_VAR

SUPER^();
Yst_Izm_trig(clk:=((Yst_izm <> Yst_T1) 	AND (Yst_izm >= 3) AND (Yst_izm < 100)));
IF 	Yst_Izm_trig.Q THEN
	Yst_T1 := Yst_izm;
	SaveToFile();
END_IF	
Yst_First_izm(clk:=((Yst_izm = 0) AND (Yst_T1 = 0) AND flag));
IF	Yst_First_izm.Q	THEN
	Yst_T1 := 3;
	Yst_izm := Yst_T1;
	SaveToFile();
END_IF;
flag:=TRUE;

METHOD PROTECTED readPersistent
VAR_INPUT
END_VAR

Yst_izm:=STRING_TO_uint(readValue());
END_METHOD

METHOD PROTECTED writePersistent
VAR_INPUT
END_VAR

writeValue(value:= uint_TO_STRING(Yst_T1),'Наработка');
END_METHOD

END_FUNCTION_BLOCK

// K2/std12k5/Ystavki/Tvkl_AVOM1
	{attribute 'symbol' := 'none'}
FUNCTION_BLOCK Tvkl_AVOM1 EXTENDS Baseobject
VAR_INPUT
	{attribute 'symbol' := 'readwright'}
	Yst_izm:UINT;
END_VAR
VAR_OUTPUT
	{attribute 'symbol' := 'read'}
	Yst_T1:UINT;
	
END_VAR
VAR
	flag:BOOL;
	Yst_Izm_trig:R_TRIG;
	Yst_First_izm:R_TRIG;
END_VAR

SUPER^();
Yst_Izm_trig(clk:=((Yst_izm <> Yst_T1) 	AND (Yst_izm >= 3) AND (Yst_izm < 100)));
IF 	Yst_Izm_trig.Q THEN
	Yst_T1 := Yst_izm;
	SaveToFile();
END_IF	
Yst_First_izm(clk:=((Yst_izm = 0) AND (Yst_T1 = 0) AND flag));
IF	Yst_First_izm.Q	THEN
	Yst_T1 := 3;
	Yst_izm := Yst_T1;
	SaveToFile();
END_IF;
flag:=TRUE;

METHOD PROTECTED readPersistent
VAR_INPUT
END_VAR

Yst_izm:=STRING_TO_uint(readValue());
END_METHOD

METHOD PROTECTED writePersistent
VAR_INPUT
END_VAR

writeValue(value:= uint_TO_STRING(Yst_T1),'Наработка');
END_METHOD

END_FUNCTION_BLOCK

// K1/std12k5/Ystavki/Tvkl_AVOM2
	{attribute 'symbol' := 'none'}
FUNCTION_BLOCK Tvkl_AVOM2 EXTENDS Baseobject
VAR_INPUT
	{attribute 'symbol' := 'readwright'}
	Yst_izm:UINT;
END_VAR
VAR_OUTPUT
	{attribute 'symbol' := 'read'}
	Yst_T2:UINT;
	
END_VAR
VAR
	flag:BOOL;
	Yst_Izm_trig:R_TRIG;
	Yst_First_izm:R_TRIG;
END_VAR

SUPER^();
Yst_Izm_trig(clk:=((Yst_izm <> Yst_T2) 	AND (Yst_izm >=3) AND (Yst_izm < 100)));
IF 	Yst_Izm_trig.Q	THEN
	Yst_T2 := Yst_izm;
	SaveToFile();
END_IF	
Yst_First_izm(clk:=((Yst_izm = 0) AND (Yst_T2 = 0) AND flag));
IF	Yst_First_izm.Q  THEN
	Yst_T2 := 3;
	Yst_izm := Yst_T2;
	SaveToFile();
END_IF;
flag:=TRUE;

METHOD PROTECTED readPersistent
VAR_INPUT
END_VAR

Yst_izm:=STRING_TO_uint(readValue());
END_METHOD

METHOD PROTECTED writePersistent
VAR_INPUT
END_VAR

writeValue(value:= uint_TO_STRING(Yst_T2),'Наработка');
END_METHOD

END_FUNCTION_BLOCK

// K2/std12k5/Ystavki/Tvkl_AVOM2
	{attribute 'symbol' := 'none'}
FUNCTION_BLOCK Tvkl_AVOM2 EXTENDS Baseobject
VAR_INPUT
	{attribute 'symbol' := 'readwright'}
	Yst_izm:UINT;
END_VAR
VAR_OUTPUT
	{attribute 'symbol' := 'read'}
	Yst_T2:UINT;
	
END_VAR
VAR
	flag:BOOL;
	Yst_Izm_trig:R_TRIG;
	Yst_First_izm:R_TRIG;
END_VAR

SUPER^();
Yst_Izm_trig(clk:=((Yst_izm <> Yst_T2) 	AND (Yst_izm >=3) AND (Yst_izm < 100)));
IF 	Yst_Izm_trig.Q	THEN
	Yst_T2 := Yst_izm;
	SaveToFile();
END_IF	
Yst_First_izm(clk:=((Yst_izm = 0) AND (Yst_T2 = 0) AND flag));
IF	Yst_First_izm.Q  THEN
	Yst_T2 := 3;
	Yst_izm := Yst_T2;
	SaveToFile();
END_IF;
flag:=TRUE;

METHOD PROTECTED readPersistent
VAR_INPUT
END_VAR

Yst_izm:=STRING_TO_uint(readValue());
END_METHOD

METHOD PROTECTED writePersistent
VAR_INPUT
END_VAR

writeValue(value:= uint_TO_STRING(Yst_T2),'Наработка');
END_METHOD

END_FUNCTION_BLOCK

// K1/std12k5/Ystavki/Tvkl_AVOM3
	{attribute 'symbol' := 'none'}
FUNCTION_BLOCK Tvkl_AVOM3 EXTENDS Baseobject
VAR_INPUT
	{attribute 'symbol' := 'readwright'}
	Yst_izm:UINT;
END_VAR
VAR_OUTPUT
	{attribute 'symbol' := 'read'}
	Yst_T3:UINT;
	
END_VAR
VAR
	flag:BOOL;
	Yst_Izm_trig:R_TRIG;
	Yst_First_izm:R_TRIG;
END_VAR

SUPER^();
Yst_Izm_trig(clk:=((Yst_izm <> Yst_T3) 	AND (Yst_izm >=3) AND (Yst_izm < 100)));
IF 	Yst_Izm_trig.Q THEN
	Yst_T3 := Yst_izm;
	SaveToFile();
END_IF	
Yst_First_izm(clk:=((Yst_izm = 0) AND (Yst_T3 = 0) AND flag));
IF	Yst_First_izm.Q THEN
	Yst_T3 := 3;
	Yst_izm := Yst_T3;
	SaveToFile();
END_IF;



flag:=TRUE;

METHOD PROTECTED readPersistent
VAR_INPUT
END_VAR

Yst_izm:=STRING_TO_uint(readValue());
END_METHOD

METHOD PROTECTED writePersistent
VAR_INPUT
END_VAR

writeValue(value:= uint_TO_STRING(Yst_T3),'Наработка');
END_METHOD

END_FUNCTION_BLOCK

// K2/std12k5/Ystavki/Tvkl_AVOM3
	{attribute 'symbol' := 'none'}
FUNCTION_BLOCK Tvkl_AVOM3 EXTENDS Baseobject
VAR_INPUT
	{attribute 'symbol' := 'readwright'}
	Yst_izm:UINT;
END_VAR
VAR_OUTPUT
	{attribute 'symbol' := 'read'}
	Yst_T3:UINT;
	
END_VAR
VAR
	flag:BOOL;
	Yst_Izm_trig:R_TRIG;
	Yst_First_izm:R_TRIG;
END_VAR

SUPER^();
Yst_Izm_trig(clk:=((Yst_izm <> Yst_T3) 	AND (Yst_izm >=3) AND (Yst_izm < 100)));
IF 	Yst_Izm_trig.Q THEN
	Yst_T3 := Yst_izm;
	SaveToFile();
END_IF	
Yst_First_izm(clk:=((Yst_izm = 0) AND (Yst_T3 = 0) AND flag));
IF	Yst_First_izm.Q THEN
	Yst_T3 := 3;
	Yst_izm := Yst_T3;
	SaveToFile();
END_IF;



flag:=TRUE;

METHOD PROTECTED readPersistent
VAR_INPUT
END_VAR

Yst_izm:=STRING_TO_uint(readValue());
END_METHOD

METHOD PROTECTED writePersistent
VAR_INPUT
END_VAR

writeValue(value:= uint_TO_STRING(Yst_T3),'Наработка');
END_METHOD

END_FUNCTION_BLOCK

// K1/std12k5/Ystavki/Tvkl_AVOM4
	{attribute 'symbol' := 'none'}
FUNCTION_BLOCK Tvkl_AVOM4 EXTENDS Baseobject
VAR_INPUT
	{attribute 'symbol' := 'readwright'}
	Yst_izm:uint;
END_VAR
VAR_OUTPUT
	{attribute 'symbol' := 'read'}
	Yst_T4:UINT;
	
END_VAR
VAR
	flag:BOOL;
	Yst_Izm_trig:R_TRIG;
	Yst_First_izm:R_TRIG;
END_VAR

SUPER^();
Yst_Izm_trig(clk:=((Yst_izm <> Yst_T4) AND (Yst_izm >= 3) AND (Yst_izm < 100)));
IF 	Yst_Izm_trig.Q THEN
	Yst_T4 := Yst_izm;
	SaveToFile ();
END_IF	
Yst_First_izm(clk:=((Yst_izm = 0) AND (Yst_T4 = 0) AND flag));
IF	Yst_First_izm.Q THEN
	Yst_T4 := 3;
	Yst_izm := Yst_T4;
	SaveToFile();
END_IF;
flag:=TRUE;

METHOD PROTECTED readPersistent
VAR_INPUT
END_VAR

Yst_izm:=STRING_TO_uint(readValue());
END_METHOD

METHOD PROTECTED writePersistent
VAR_INPUT
END_VAR

writeValue(value:= uint_TO_STRING(Yst_T4),'Наработка');
END_METHOD

END_FUNCTION_BLOCK

// K2/std12k5/Ystavki/Tvkl_AVOM4
	{attribute 'symbol' := 'none'}
FUNCTION_BLOCK Tvkl_AVOM4 EXTENDS Baseobject
VAR_INPUT
	{attribute 'symbol' := 'readwright'}
	Yst_izm:uint;
END_VAR
VAR_OUTPUT
	{attribute 'symbol' := 'read'}
	Yst_T4:UINT;
	
END_VAR
VAR
	flag:BOOL;
	Yst_Izm_trig:R_TRIG;
	Yst_First_izm:R_TRIG;
END_VAR

SUPER^();
Yst_Izm_trig(clk:=((Yst_izm <> Yst_T4) AND (Yst_izm >= 3) AND (Yst_izm < 100)));
IF 	Yst_Izm_trig.Q THEN
	Yst_T4 := Yst_izm;
	SaveToFile ();
END_IF	
Yst_First_izm(clk:=((Yst_izm = 0) AND (Yst_T4 = 0) AND flag));
IF	Yst_First_izm.Q THEN
	Yst_T4 := 3;
	Yst_izm := Yst_T4;
	SaveToFile();
END_IF;
flag:=TRUE;

METHOD PROTECTED readPersistent
VAR_INPUT
END_VAR

Yst_izm:=STRING_TO_uint(readValue());
END_METHOD

METHOD PROTECTED writePersistent
VAR_INPUT
END_VAR

writeValue(value:= uint_TO_STRING(Yst_T4),'Наработка');
END_METHOD

END_FUNCTION_BLOCK

// K1/std12k5/Ystavki/Tvykl_AVOM1
	{attribute 'symbol' := 'none'}
FUNCTION_BLOCK Tvykl_AVOM1 EXTENDS Baseobject
VAR_INPUT
	{attribute 'symbol' := 'readwright'}
	Yst_izm:uint;
END_VAR
VAR_OUTPUT
	{attribute 'symbol' := 'read'}
	Yst_T1:UINT;
	
END_VAR
VAR
	flag:BOOL;
	Yst_Izm_trig:R_TRIG;
	Yst_First_izm:R_TRIG;
END_VAR

SUPER^();
Yst_Izm_trig(clk:=((Yst_izm <> Yst_T1) AND (Yst_izm > 0) AND (Yst_izm < 100)));
IF 	Yst_Izm_trig.Q THEN
	Yst_T1 := Yst_izm;
	SaveToFile();

END_IF	
Yst_First_izm(clk:=((Yst_izm = 0) AND (Yst_T1 = 0) AND flag));
IF	Yst_First_izm.Q  THEN
	Yst_T1 := 3;
	Yst_izm := Yst_T1;
	SaveToFile();
END_IF;



flag:=TRUE;

METHOD PROTECTED readPersistent
VAR_INPUT
END_VAR

Yst_izm:=STRING_TO_uint(readValue());
END_METHOD

METHOD PROTECTED writePersistent
VAR_INPUT
END_VAR

writeValue(value:= uint_TO_STRING(Yst_T1),'Наработка');
END_METHOD

END_FUNCTION_BLOCK

// K2/std12k5/Ystavki/Tvykl_AVOM1
	{attribute 'symbol' := 'none'}
FUNCTION_BLOCK Tvykl_AVOM1 EXTENDS Baseobject
VAR_INPUT
	{attribute 'symbol' := 'readwright'}
	Yst_izm:uint;
END_VAR
VAR_OUTPUT
	{attribute 'symbol' := 'read'}
	Yst_T1:UINT;
	
END_VAR
VAR
	flag:BOOL;
	Yst_Izm_trig:R_TRIG;
	Yst_First_izm:R_TRIG;
END_VAR

SUPER^();
Yst_Izm_trig(clk:=((Yst_izm <> Yst_T1) AND (Yst_izm > 0) AND (Yst_izm < 100)));
IF 	Yst_Izm_trig.Q THEN
	Yst_T1 := Yst_izm;
	SaveToFile();

END_IF	
Yst_First_izm(clk:=((Yst_izm = 0) AND (Yst_T1 = 0) AND flag));
IF	Yst_First_izm.Q  THEN
	Yst_T1 := 3;
	Yst_izm := Yst_T1;
	SaveToFile();
END_IF;



flag:=TRUE;

METHOD PROTECTED readPersistent
VAR_INPUT
END_VAR

Yst_izm:=STRING_TO_uint(readValue());
END_METHOD

METHOD PROTECTED writePersistent
VAR_INPUT
END_VAR

writeValue(value:= uint_TO_STRING(Yst_T1),'Наработка');
END_METHOD

END_FUNCTION_BLOCK

// K1/std12k5/Ystavki/Tvykl_AVOM2
	{attribute 'symbol' := 'none'}
FUNCTION_BLOCK Tvykl_AVOM2 EXTENDS Baseobject
VAR_INPUT
	{attribute 'symbol' := 'readwright'}
	Yst_izm:uint;
END_VAR
VAR_OUTPUT
	{attribute 'symbol' := 'read'}
	Yst_T2:UINT;
	
END_VAR
VAR
	flag:BOOL;
	Yst_Izm_trig:R_TRIG;
	Yst_First_izm:R_TRIG;
END_VAR

SUPER^();
Yst_Izm_trig(clk:=((Yst_izm <> Yst_T2) 	AND (Yst_izm > 0) AND (Yst_izm < 100)));
IF 	Yst_Izm_trig.Q THEN
	Yst_T2 := Yst_izm;
	SaveToFile();

END_IF	
Yst_First_izm(clk:=((Yst_izm = 0) AND (Yst_T2 = 0) AND flag ));
IF	Yst_First_izm.Q THEN
	Yst_T2 := 3;
	Yst_izm := Yst_T2;
	SaveToFile();
END_IF;


flag:=TRUE;

METHOD PROTECTED readPersistent
VAR_INPUT
END_VAR

Yst_izm:=STRING_TO_uint(readValue());
END_METHOD

METHOD PROTECTED writePersistent
VAR_INPUT
END_VAR

writeValue(value:= uint_TO_STRING(Yst_T2),'Наработка');
END_METHOD

END_FUNCTION_BLOCK

// K2/std12k5/Ystavki/Tvykl_AVOM2
	{attribute 'symbol' := 'none'}
FUNCTION_BLOCK Tvykl_AVOM2 EXTENDS Baseobject
VAR_INPUT
	{attribute 'symbol' := 'readwright'}
	Yst_izm:uint;
END_VAR
VAR_OUTPUT
	{attribute 'symbol' := 'read'}
	Yst_T2:UINT;
	
END_VAR
VAR
	flag:BOOL;
	Yst_Izm_trig:R_TRIG;
	Yst_First_izm:R_TRIG;
END_VAR

SUPER^();
Yst_Izm_trig(clk:=((Yst_izm <> Yst_T2) 	AND (Yst_izm > 0) AND (Yst_izm < 100)));
IF 	Yst_Izm_trig.Q THEN
	Yst_T2 := Yst_izm;
	SaveToFile();

END_IF	
Yst_First_izm(clk:=((Yst_izm = 0) AND (Yst_T2 = 0) AND flag ));
IF	Yst_First_izm.Q THEN
	Yst_T2 := 3;
	Yst_izm := Yst_T2;
	SaveToFile();
END_IF;


flag:=TRUE;

METHOD PROTECTED readPersistent
VAR_INPUT
END_VAR

Yst_izm:=STRING_TO_uint(readValue());
END_METHOD

METHOD PROTECTED writePersistent
VAR_INPUT
END_VAR

writeValue(value:= uint_TO_STRING(Yst_T2),'Наработка');
END_METHOD

END_FUNCTION_BLOCK

// K1/std12k5/Ystavki/Tvykl_AVOM3
	{attribute 'symbol' := 'none'}
FUNCTION_BLOCK Tvykl_AVOM3 EXTENDS Baseobject
VAR_INPUT
	{attribute 'symbol' := 'readwright'}
	Yst_izm:uint;
END_VAR
VAR_OUTPUT
	{attribute 'symbol' := 'read'}
	Yst_T3:UINT;
	
END_VAR
VAR
	flag:BOOL;
	Yst_Izm_trig:R_TRIG;
	Yst_First_izm:R_TRIG;
END_VAR

SUPER^();
Yst_Izm_trig(clk:=((Yst_izm <> Yst_T3) AND (Yst_izm > 0) AND (Yst_izm < 100)));
IF 	Yst_Izm_trig.Q THEN
	Yst_T3 := Yst_izm;
	SaveToFile();

END_IF	
Yst_First_izm(clk:=((Yst_izm = 0) AND (Yst_T3 = 0) AND flag));
IF	Yst_First_izm.Q THEN
	Yst_T3 := 3;
	Yst_izm := Yst_T3;
	SaveToFile();
END_IF;
flag:=TRUE;

METHOD PROTECTED readPersistent
VAR_INPUT
END_VAR

Yst_izm:=STRING_TO_uint(readValue());
END_METHOD

METHOD PROTECTED writePersistent
VAR_INPUT
END_VAR

writeValue(value:= uint_TO_STRING(Yst_T3),'Наработка');
END_METHOD

END_FUNCTION_BLOCK

// K2/std12k5/Ystavki/Tvykl_AVOM3
	{attribute 'symbol' := 'none'}
FUNCTION_BLOCK Tvykl_AVOM3 EXTENDS Baseobject
VAR_INPUT
	{attribute 'symbol' := 'readwright'}
	Yst_izm:uint;
END_VAR
VAR_OUTPUT
	{attribute 'symbol' := 'read'}
	Yst_T3:UINT;
	
END_VAR
VAR
	flag:BOOL;
	Yst_Izm_trig:R_TRIG;
	Yst_First_izm:R_TRIG;
END_VAR

SUPER^();
Yst_Izm_trig(clk:=((Yst_izm <> Yst_T3) AND (Yst_izm > 0) AND (Yst_izm < 100)));
IF 	Yst_Izm_trig.Q THEN
	Yst_T3 := Yst_izm;
	SaveToFile();

END_IF	
Yst_First_izm(clk:=((Yst_izm = 0) AND (Yst_T3 = 0) AND flag));
IF	Yst_First_izm.Q THEN
	Yst_T3 := 3;
	Yst_izm := Yst_T3;
	SaveToFile();
END_IF;
flag:=TRUE;

METHOD PROTECTED readPersistent
VAR_INPUT
END_VAR

Yst_izm:=STRING_TO_uint(readValue());
END_METHOD

METHOD PROTECTED writePersistent
VAR_INPUT
END_VAR

writeValue(value:= uint_TO_STRING(Yst_T3),'Наработка');
END_METHOD

END_FUNCTION_BLOCK

// K1/std12k5/Ystavki/Tvykl_AVOM4
	{attribute 'symbol' := 'none'}
FUNCTION_BLOCK Tvykl_AVOM4 EXTENDS Baseobject
VAR_INPUT
	{attribute 'symbol' := 'readwright'}
	Yst_izm:uint;
END_VAR
VAR_OUTPUT
	{attribute 'symbol' := 'read'}
	Yst_T4:UINT;
	
END_VAR
VAR
	flag:BOOL;
	Yst_Izm_trig:R_TRIG;
	Yst_First_izm:R_TRIG;
END_VAR

SUPER^();
Yst_Izm_trig(clk:=((Yst_izm <> Yst_T4) AND (Yst_izm > 0) AND (Yst_izm < 100)));
IF 	Yst_Izm_trig.Q THEN
	Yst_T4 := Yst_izm;
	SaveToFile();

END_IF	
Yst_First_izm(clk:=((Yst_izm = 0) AND (Yst_T4 = 0) AND flag));
IF	Yst_First_izm.Q THEN
	Yst_T4 := 3;
	Yst_izm := Yst_T4;
	SaveToFile();
END_IF;

flag:=true;

METHOD PROTECTED readPersistent
VAR_INPUT
END_VAR

Yst_izm:=STRING_TO_uint(readValue());
END_METHOD

METHOD PROTECTED writePersistent
VAR_INPUT
END_VAR

writeValue(value:= uint_TO_STRING(Yst_T4),'Наработка');
END_METHOD

END_FUNCTION_BLOCK

// K2/std12k5/Ystavki/Tvykl_AVOM4
	{attribute 'symbol' := 'none'}
FUNCTION_BLOCK Tvykl_AVOM4 EXTENDS Baseobject
VAR_INPUT
	{attribute 'symbol' := 'readwright'}
	Yst_izm:uint;
END_VAR
VAR_OUTPUT
	{attribute 'symbol' := 'read'}
	Yst_T4:UINT;
	
END_VAR
VAR
	flag:BOOL;
	Yst_Izm_trig:R_TRIG;
	Yst_First_izm:R_TRIG;
END_VAR

SUPER^();
Yst_Izm_trig(clk:=((Yst_izm <> Yst_T4) AND (Yst_izm > 0) AND (Yst_izm < 100)));
IF 	Yst_Izm_trig.Q THEN
	Yst_T4 := Yst_izm;
	SaveToFile();

END_IF	
Yst_First_izm(clk:=((Yst_izm = 0) AND (Yst_T4 = 0) AND flag));
IF	Yst_First_izm.Q THEN
	Yst_T4 := 3;
	Yst_izm := Yst_T4;
	SaveToFile();
END_IF;

flag:=true;

METHOD PROTECTED readPersistent
VAR_INPUT
END_VAR

Yst_izm:=STRING_TO_uint(readValue());
END_METHOD

METHOD PROTECTED writePersistent
VAR_INPUT
END_VAR

writeValue(value:= uint_TO_STRING(Yst_T4),'Наработка');
END_METHOD

END_FUNCTION_BLOCK

// K1/std12k5/Narabotka/Work
	{attribute 'symbol' := 'none'}
FUNCTION_BLOCK work EXTENDS BaseIM
VAR_INPUT
END_VAR
VAR_OUTPUT
	
		{attribute 'symbol' := 'read'}
	narabotka:UDINT;
	narabotka_:ExtNarabotka (table:=ADR (objectTable)):=(saveInterval:=T#1H);
END_VAR
VAR
(*timer:RTC;	
	saveTimer:TON:=(PT:=T#600S);
	Narabotka_hour:R_TRIG;
	AvomStartted:R_TRIG;
	narabotka_Izm:UDINT;*)
END_VAR

SUPER^();
narabotka_.started:=((algmanager.mode=modegpa.MODE_WORK_K) OR (algmanager.mode=modegpa.MODE_WORK_M));
narabotka:=(narabotka_.narabotka/3600);

(*


AvomStartted(CLK:=((algmanager.mode=modegpa.MODE_WORK_K) OR (algmanager.mode=modegpa.MODE_WORK_M)));

	timer.PDT:=UDINT_TO_DT(narabotka_izm);

IF ((algmanager.mode=modegpa.MODE_WORK_K) OR (algmanager.mode=modegpa.MODE_WORK_M)) THEN
	narabotka_izm:=DT_TO_UDINT( timer.CDT);
	timer.EN:=TRUE;
ELSE
	timer.EN:=FALSE;
END_IF
narabotka_hour (clk:=(narabotka_izm >=3600));
IF	narabotka_hour.Q THEN
	narabotka:=narabotka+1;
	timer.EN:=FALSE;
	narabotka_izm:=0;
END_IF
timer();

saveTimer(IN:=true);
IF saveTimer.Q THEN
	SaveToFile();
	saveTimer(IN:=FALSE);
END_IF*)

METHOD PROTECTED readPersistent
VAR_INPUT
END_VAR

narabotka:=STRING_TO_UDINT(readValue());
narabotka_izm:=STRING_TO_UDINT(readValue());
END_METHOD

METHOD PROTECTED writePersistent
VAR_INPUT
END_VAR

writeValue(value:= UDINT_TO_STRING(narabotka),'Наработка');
writeValue(value:= UDINT_TO_STRING(narabotka_izm),'Наработка_izm');
END_METHOD

END_FUNCTION_BLOCK

// K2/std12k5/Natabotka/Work
	{attribute 'symbol' := 'none'}
FUNCTION_BLOCK work EXTENDS BaseIM
VAR_INPUT
END_VAR
VAR_OUTPUT
	
		{attribute 'symbol' := 'read'}
	narabotka:UDINT;
	narabotka_:ExtNarabotka (table:=ADR (objectTable)):=(saveInterval:=T#1H);
END_VAR
VAR
(*timer:RTC;	
	saveTimer:TON:=(PT:=T#600S);
	Narabotka_hour:R_TRIG;
	AvomStartted:R_TRIG;
	narabotka_Izm:UDINT;*)
END_VAR

SUPER^();
narabotka_.started:=((algmanager.mode=modegpa.MODE_WORK_K) OR (algmanager.mode=modegpa.MODE_WORK_M));
narabotka:=(narabotka_.narabotka/3600);

(*

AvomStartted(CLK:=((algmanager.mode=modegpa.MODE_WORK_K) OR (algmanager.mode=modegpa.MODE_WORK_M)));

	timer.PDT:=UDINT_TO_DT(narabotka_izm);

IF ((algmanager.mode=modegpa.MODE_WORK_K) OR (algmanager.mode=modegpa.MODE_WORK_M)) THEN
	narabotka_izm:=DT_TO_UDINT( timer.CDT);
	timer.EN:=TRUE;
ELSE
	timer.EN:=FALSE;
END_IF
narabotka_hour (clk:=(narabotka_izm >=3600));
IF	narabotka_hour.Q THEN
	narabotka:=narabotka+1;
	timer.EN:=FALSE;
	narabotka_izm:=0;
END_IF
timer();

saveTimer(IN:=true);
IF saveTimer.Q THEN
	SaveToFile();
	saveTimer(IN:=FALSE);
END_IF*)

METHOD PROTECTED readPersistent
VAR_INPUT
END_VAR

narabotka:=STRING_TO_UDINT(readValue());
narabotka_izm:=STRING_TO_UDINT(readValue());
END_METHOD

METHOD PROTECTED writePersistent
VAR_INPUT
END_VAR

writeValue(value:= UDINT_TO_STRING(narabotka),'Наработка');
writeValue(value:= UDINT_TO_STRING(narabotka_izm),'Наработка_izm');
END_METHOD

END_FUNCTION_BLOCK

// LowLevel_Algoritms/Common/everifingTrue
	{attribute 'symbol' := 'none'}
FUNCTION_BLOCK everifingTrue EXTENDS DISource
VAR_INPUT
END_VAR
VAR_OUTPUT
	DO_kr6:BOOL;
	DO_kr6A:BOOL;
END_VAR
VAR
END_VAR

SUPER^();
imit:=TRUE;
reliability:=65535;
value:=65535;

END_FUNCTION_BLOCK

// LowLevel_Algoritms/im/IMs
{attribute 'symbol' := 'none'}
FUNCTION_BLOCK IMs EXTENDS BaseIM
VAR_INPUT
	di1:REFERENCE TO reliablebit;
	di2:REFERENCE TO reliablebit;
END_VAR 
VAR_OUTPUT
END_VAR
VAR
END_VAR

SUPER^();
IF __ISVALIDREF(di1) AND __ISVALIDREF(di2) THEN
	IF	(di1.value = 0) AND  (di2.reliability = 1) THEN
		statusSet.setBit (bitNum:=0,value:=1);
	ELSE
		statusSet.setBit (bitNum:=0,value:=0);
	END_IF
END_IF

END_FUNCTION_BLOCK

// LowLevel_Algoritms/im/Krans_Sdvig
{attribute 'symbol' := 'none'}
FUNCTION_BLOCK Krans_Sdvig EXTENDS BaseIm
VAR_INPUT
	Krans:REFERENCE TO Kran;
	block:REFERENCE TO DiscretParametr(*(table:=ADR(objectTable))*);
END_VAR
VAR_OUTPUT
END_VAR
VAR
	Kran_state:statusDualInput;
	Trig:R_TRIG;
END_VAR

SUPER^();
Trig (clk:=(block.Value = 1));
IF __ISVALIDREF(Krans) THEN
	IF (krans.onStatus <> Kran_state) AND krans.sdvig AND  (block.Value = 0)	THEN
		statusSet.setBit (bitNum:=0,value:=1);
		IF	Kran_state = statusDualInput.status_on THEN
			Krans.on ();
		END_IF
		IF	Kran_state = statusDualInput.status_off THEN
			Krans.off ();
		END_IF
	ELSE 
		statusSet.setBit (bitNum:=0,value:=0);
		IF	Trig.Q THEN
			Kran_state:=krans.onStatus;
			krans.reset ();
		END_IF
	END_IF
	IF	(krans.onStatus = statusDualInput.status_on)  OR (krans.onStatus = statusDualInput.status_off) THEN
		Kran_state:=krans.onStatus;
	END_IF;
END_IF

END_FUNCTION_BLOCK

// LowLevel_Algoritms/im/NasosNu
	{attribute 'symbol' := 'none'}
FUNCTION_BLOCK NasosNu EXTENDS Nasos
VAR_INPUT
		{attribute 'symbol' := 'read'}
	nu1:Nasos(table:=ADR(objectTable));//{name:НУ1}	
		{attribute 'symbol' := 'read'}
	nu2:Nasos(table:=ADR(objectTable));//{name:НУ2}	
	
		
END_VAR

VAR_OUTPUT
		{attribute 'symbol' := 'readwrite'}
	mainNasos:DiscretParametr(table:=ADR(objectTable));//{name:Номер основного насоса}
END_VAR
VAR
	changevalue:WORD;
	Changevalue_trig : R_trig;
END_VAR
VAR CONSTANT
END_VAR

SUPER^();

IF	algoritms.autoNu_1.flag1 OR algoritms.autoNu_2.flag1 THEN
	mainNasos.setValue (0);
END_IF
IF	algoritms.autoNu_1.flag2 OR algoritms.autoNu_2.flag2 THEN
	mainNasos.setValue (1);
END_IF
Changevalue_trig (Clk:= algoritms.autoNu_2.flag3);
IF	Changevalue_trig.Q THEN
	changevalue:=mainNasos.Value;
END_IF
IF	algoritms.autoNu_2.flag3 THEN
	mainNasos.setValue	(changevalue);
END_IF
IF	(nu1.onStatus = statusDualInput.STATUS_OFF) AND (nu2.onStatus = statusDualInput.STATUS_OFF) THEN
	onStatus := statusDualInput.STATUS_OFF;
END_IF
IF	algoritms.autoNu_1.flag1 OR algoritms.autoNu_2.flag1 OR algoritms.autoNu_1.flag2 OR algoritms.autoNu_2.flag2 OR algoritms.autoNu_2.flag3 THEN
	mainNasos.DisableOpcControl ();
ELSE
	mainNasos.EnableOpcControl ();
END_IF

METHOD PUBLIC Off
VAR_INPUT
END_VAR
SUPER^();
nu1.off();
nu2.off ();
END_METHOD

END_FUNCTION_BLOCK

// K1/std12k5/nasos/AutoAVOM
	{attribute 'symbol' := 'none'}
FUNCTION_BLOCK  AutoAVOM EXTENDS BaseAlgoritm
VAR_INPUT
	T_posle_AVOM :REFERENCE TO AiSource;
	A1:REFERENCE TO Avom1;
	A2:REFERENCE TO Avom2;
	A3:REFERENCE TO Avom3;
	A4:REFERENCE TO Avom4;
END_VAR
VAR_OUTPUT
	flag_vkl1:BOOL;
	flag_vkl2:BOOL;
	flag_vkl3:BOOL;
	flag_vkl4:BOOL;
	i: UINT;
	num_vykl:UINT;
	num_arr:ARRAY[0..3] OF UINT;
	Num:UINT;
	
	T1_vklAVOM:TON;
	T2_vklAVOM:TON;
	T3_vklAVOM:TON;
	T4_vklAVOM:TON;
	T1_vyklAVOM:TON;
	T2_vyklAVOM:TON;
	T3_vyklAVOM:TON;
	T4_vyklAVOM:TON;
	
	Vkl_AVOM1:R_TRIG;
	Vkl_AVOM2:R_TRIG;
	Vkl_AVOM3:R_TRIG;
	Vkl_AVOM4:R_TRIG;
	
	Vykl_AVOM1:R_TRIG;
	Vykl_AVOM2:R_TRIG;
	Vykl_AVOM3:R_TRIG;
	Vykl_AVOM4:R_TRIG;
END_VAR
VAR
	i1_izm:UINT;
	i2_izm:UINT;
	
	
END_VAR

SUPER^();
T1_vklAVOM(IN:=((T_posle_AVOM.interval>=statusAi.NORmaL) AND (T_posle_AVOM.value >= Ystavki.Yst_AVOM_T1.Yst_T1) AND NOT flag_vkl1), PT:=UINT_TO_TIME (Ystavki.Yst_Tvkl_AVOM1.Yst_T1 * 1000) );
Vkl_AVOM1 (CLK:=(T1_vklAVOM.Q ));
IF	Vkl_AVOM1.Q THEN
	flag_vkl1:=TRUE;
	CASE (num) OF
	4:	IF (num_arr 	[0] =0) THEN
			num:=1;
			num_arr 	[0]:=1;
		END_IF
	0..3:	num_arr 	[num]:= 1;
			num 		:= num + 1;
	END_CASE
	avoms_vkl ();
END_IF
/////////////////////////////////////////////////////////////////////
T2_vklAVOM(IN:=((T_posle_AVOM.interval>=statusAi.NORmaL) AND (T_posle_AVOM.value >= Ystavki.Yst_AVOM_T2.Yst_T2) AND flag_vkl1 AND NOT flag_vkl2), PT:=UINT_TO_TIME (Ystavki.Yst_Tvkl_AVOM2.Yst_T2 * 1000));
Vkl_AVOM2 (CLK:=(T2_vklAVOM.Q ));
IF	Vkl_AVOM2.Q THEN
	flag_vkl2:=TRUE;
	CASE (num) OF
	4:	IF (num_arr 	[0] =0) THEN
			num:=1;
			num_arr 	[0]:=2;
		END_IF
	0..3:	num_arr 	[num]:= 2;
			num 		:= num + 1;
	END_CASE
	avoms_vkl ();
END_IF
/////////////////////////////////////////////////////////////////////
T3_vklAVOM(IN:=((T_posle_AVOM.interval>=statusAi.NORmaL) AND (T_posle_AVOM.value >= Ystavki.Yst_AVOM_T3.Yst_T3) AND flag_vkl1 AND flag_vkl2 AND NOT flag_vkl3), PT:=UINT_TO_TIME (Ystavki.Yst_Tvkl_AVOM3.Yst_T3 * 1000));
Vkl_AVOM3 (CLK:=(T3_vklAVOM.Q ));
IF	Vkl_AVOM3.Q THEN
	flag_vkl3:=TRUE;
	CASE (num) OF
	4:	IF (num_arr 	[0] =0) THEN
			num:=1;
			num_arr 	[0]:=3;
		END_IF
	0..3:	num_arr 	[num]:= 3;
			num 		:= num + 1;
	END_CASE
	avoms_vkl ();
END_IF
/////////////////////////////////////////////////////////////////////
T4_vklAVOM(IN:=((T_posle_AVOM.interval>=statusAi.NORmaL) AND (T_posle_AVOM.value >= Ystavki.Yst_AVOM_T4.Yst_T4) AND flag_vkl3 AND flag_vkl1 AND flag_vkl2 AND NOT flag_vkl4 ), PT:=UINT_TO_TIME (Ystavki.Yst_Tvkl_AVOM4.Yst_T4 * 1000));
Vkl_AVOM4 (CLK:=(T4_vklAVOM.Q ));
IF	Vkl_AVOM4.Q THEN
	flag_vkl4:=TRUE;
	CASE (num) OF
	4:	IF (num_arr 	[0] =0) THEN
			num:=1;
			num_arr 	[0]:=4;
		END_IF
	0..3:	num_arr 	[num]:= 4;
			num 		:= num + 1;
	END_CASE
	avoms_vkl ();
END_IF
/////////////////////////////////////////////////////////////////////

T1_vyklAVOM(IN:=((T_posle_AVOM.interval>=statusAi.NORmaL) AND (T_posle_AVOM.value <= (Ystavki.Yst_AVOM_T1.Yst_T1 - Ystavki.Yst_DTvykl_AVOM1.Yst_T1)) AND flag_vkl1 AND NOT flag_vkl2), PT:=UINT_TO_TIME (Ystavki.Yst_Tvykl_AVOM1.Yst_T1 * 1000));
Vykl_AVOM1 (CLK:=(T1_vyklAVOM.Q ));
IF	Vykl_AVOM1.Q THEN
	flag_vkl1:=FALSE;
	FOR i:=0 TO 3 DO
		IF 	num_arr [i] > 0 THEN
			num_arr [i] := num_arr [i] - 1;
		END_IF
		IF 	num_arr [i] = 0 THEN
			CASE i OF
				0: num_vykl:= 1;
				1: num_vykl:= 2;
				2: num_vykl:= 3;
				3: num_vykl:= 4;
			END_CASE
			avoms_vykl ();
		END_IF
	END_FOR
	avoms_vykl ();
END_IF
/////////////////////////////////////////////////////////////////////
T2_vyklAVOM(IN:=((T_posle_AVOM.interval>=statusAi.NORmaL) AND (T_posle_AVOM.value <= (Ystavki.Yst_AVOM_T2.Yst_T2 - Ystavki.Yst_DTvykl_AVOM2.Yst_T2)) AND flag_vkl2 AND NOT flag_vkl3), PT:= UINT_TO_TIME (Ystavki.Yst_Tvykl_AVOM2.Yst_T2 * 1000));
Vykl_AVOM2 (CLK:=(T2_vyklAVOM.Q ));
IF	Vykl_AVOM2.Q THEN
	flag_vkl2:=FALSE;
	FOR i:=0 TO 3 DO
		IF 	num_arr [i] > 0 THEN
			num_arr [i] := num_arr [i] - 1;
		END_IF
		IF 	num_arr [i] = 0 THEN
			CASE i OF
				0: num_vykl:= 1;
				1: num_vykl:= 2;
				2: num_vykl:= 3;
				3: num_vykl:= 4;
			END_CASE
			avoms_vykl ();
		END_IF
	END_FOR
	avoms_vykl ();
END_IF
/////////////////////////////////////////////////////////////////////
T3_vyklAVOM(IN:=((T_posle_AVOM.interval>=statusAi.NORmaL) AND (T_posle_AVOM.value <= (Ystavki.Yst_AVOM_T3.Yst_T3 - Ystavki.Yst_DTvykl_AVOM3.Yst_T3)) AND flag_vkl3 AND NOT flag_vkl4), PT:=UINT_TO_TIME (Ystavki.Yst_Tvykl_AVOM3.Yst_T3 * 1000));
Vykl_AVOM3 (CLK:=(T3_vyklAVOM.Q ));
IF	Vykl_AVOM3.Q THEN
	flag_vkl3:=FALSE;
	FOR i:=0 TO 3 DO
		IF 	num_arr [i] > 0 THEN
			num_arr [i] := num_arr [i] - 1;
		END_IF
		IF 	num_arr [i] = 0 THEN
			CASE i OF
				0: num_vykl:= 1;
				1: num_vykl:= 2;
				2: num_vykl:= 3;
				3: num_vykl:= 4;
			END_CASE
			avoms_vykl ();
		END_IF
	END_FOR
	avoms_vykl ();
END_IF
/////////////////////////////////////////////////////////////////////
T4_vyklAVOM(IN:=((T_posle_AVOM.interval>=statusAi.NORmaL) AND (T_posle_AVOM.value <= (Ystavki.Yst_AVOM_T4.Yst_T4 - Ystavki.Yst_DTvykl_AVOM4.Yst_T4)) AND flag_vkl4 ), PT:=UINT_TO_TIME (Ystavki.Yst_Tvykl_AVOM4.Yst_T4 * 1000));
Vykl_AVOM4 (CLK:=(T4_vyklAVOM.Q ));
IF	Vykl_AVOM4.Q THEN
	flag_vkl4:=FALSE;
	FOR i:=0 TO 3 DO
		IF 	num_arr [i] > 0 THEN
			num_arr [i] := num_arr [i] - 1;
		END_IF
		IF 	num_arr [i] = 0 THEN
			CASE i OF
				0: num_vykl:= 1;
				1: num_vykl:= 2;
				2: num_vykl:= 3;
				3: num_vykl:= 4;
			END_CASE
			avoms_vykl ();
		END_IF
	END_FOR
END_IF
/////////////////////////////////////////////////////////////////////
IF	(T_posle_AVOM.interval < statusAi.NORmaL) THEN
	reset ();
END_IF

METHOD PRIVATE AVOMs_Vkl
VAR_INPUT
	
END_VAR
VAR
	
END_VAR
SUPER^();
IF	(Vkl_AVOM1.Q OR Vkl_AVOM2.Q OR Vkl_AVOM3.Q OR Vkl_AVOM4.Q) AND (num <> i1_izm)  AND (num > 0) THEN
	CASE 		Ystavki.num_Avom.Yst [num - 1] OF
		1:		A1.on ();
		2:		A2.on ();
		3:		A3.on ();
		4:		A4.on ();
		
	END_CASE
	
END_IF
i1_izm :=num;
END_METHOD

METHOD PUBLIC reset
VAR_INPUT
END_VAR
SUPER^.reset();
im.v1_Avom.off ();
im.v2_Avom.off ();
im.v3_Avom.off ();
im.v4_Avom.off ();

flag_vkl1:=FALSE;
flag_vkl2:=FALSE;
flag_vkl3:=FALSE;
flag_vkl4:=FALSE;
i:=0;
num_vykl:=0;

num_arr [0]:=0;
num_arr [1]:=0;
num_arr [2]:=0;
num_arr [3]:=0;

i1_izm:=0;
i2_izm:=0;

Num:=0;
	
T1_vklAVOM (IN:=FALSE);
T2_vklAVOM (IN:=FALSE);
T3_vklAVOM (IN:=FALSE);
T4_vklAVOM (IN:=FALSE);
	
T1_vyklAVOM (IN:=FALSE);
T2_vyklAVOM (IN:=FALSE);
T3_vyklAVOM (IN:=FALSE);
T4_vyklAVOM (IN:=FALSE);
	
Vkl_AVOM1 	(clk:=FALSE);
Vkl_AVOM2	(clk:=FALSE);
Vkl_AVOM3	(clk:=FALSE);
Vkl_AVOM4	(clk:=FALSE);
	
Vykl_AVOM1	(clk:=FALSE);
Vykl_AVOM2	(clk:=FALSE);
Vykl_AVOM3	(clk:=FALSE);
Vykl_AVOM4	(clk:=FALSE);
IF	algoritms.F2_Ch.autoAVOM_canrun_flag OR algoritms.F2_R.autoAVOM_canrun_flag THEN
	algoritms.S_AutoAVOM.CanRun:=TRUE;
	algoritms.R_AutoAVom.CanRun:=FALSE;
END_IF
END_METHOD

METHOD PRIVATE AVOMs_Vykl
VAR_INPUT
	
END_VAR
VAR
END_VAR
SUPER^();
IF	(Vykl_AVOM1.Q OR Vykl_AVOM2.Q OR Vykl_AVOM3.Q OR Vykl_AVOM4.Q) AND (num_vykl <> i2_izm)  AND (num_vykl > 0) THEN
	CASE 		Ystavki.num_Avom.Yst [num_vykl - 1] OF
		1:		A1.off ();
		2:		A2.off ();
		3:		A3.off ();
		4:		A4.off ();
	END_CASE
END_IF
i2_izm :=num_vykl;
END_METHOD

METHOD PUBLIC run
VAR_INPUT
END_VAR
SUPER^.run();
algoritms.S_AutoAVOM.CanRun:=FALSE;
algoritms.R_AutoAVom.CanRun:=TRUE;
END_METHOD

END_FUNCTION_BLOCK

// K2/std12k5/nasos/AutoAVOM
	{attribute 'symbol' := 'none'}
FUNCTION_BLOCK  AutoAVOM EXTENDS BaseAlgoritm
VAR_INPUT
	T_posle_AVOM :REFERENCE TO AiSource;
	A1:REFERENCE TO Avom1;
	A2:REFERENCE TO Avom2;
	A3:REFERENCE TO Avom3;
	A4:REFERENCE TO Avom4;
END_VAR
VAR_OUTPUT
	flag_vkl1:BOOL;
	flag_vkl2:BOOL;
	flag_vkl3:BOOL;
	flag_vkl4:BOOL;
	i: UINT;
	num_vykl:UINT;
	num_arr:ARRAY[0..3] OF UINT;
	Num:UINT;
	
	T1_vklAVOM:TON;
	T2_vklAVOM:TON;
	T3_vklAVOM:TON;
	T4_vklAVOM:TON;
	T1_vyklAVOM:TON;
	T2_vyklAVOM:TON;
	T3_vyklAVOM:TON;
	T4_vyklAVOM:TON;
	
	Vkl_AVOM1:R_TRIG;
	Vkl_AVOM2:R_TRIG;
	Vkl_AVOM3:R_TRIG;
	Vkl_AVOM4:R_TRIG;
	
	Vykl_AVOM1:R_TRIG;
	Vykl_AVOM2:R_TRIG;
	Vykl_AVOM3:R_TRIG;
	Vykl_AVOM4:R_TRIG;
END_VAR
VAR
	i1_izm:UINT;
	i2_izm:UINT;
	
	
END_VAR

SUPER^();
T1_vklAVOM(IN:=((T_posle_AVOM.interval>=statusAi.NORmaL) AND (T_posle_AVOM.value >= Ystavki.Yst_AVOM_T1.Yst_T1) AND NOT flag_vkl1), PT:=UINT_TO_TIME (Ystavki.Yst_Tvkl_AVOM1.Yst_T1 * 1000) );
Vkl_AVOM1 (CLK:=(T1_vklAVOM.Q ));
IF	Vkl_AVOM1.Q THEN
	flag_vkl1:=TRUE;
	CASE (num) OF
	4:	IF (num_arr 	[0] =0) THEN
			num:=1;
			num_arr 	[0]:=1;
		END_IF
	0..3:	num_arr 	[num]:= 1;
			num 		:= num + 1;
	END_CASE
	avoms_vkl ();
END_IF
/////////////////////////////////////////////////////////////////////
T2_vklAVOM(IN:=((T_posle_AVOM.interval>=statusAi.NORmaL) AND (T_posle_AVOM.value >= Ystavki.Yst_AVOM_T2.Yst_T2) AND flag_vkl1 AND NOT flag_vkl2), PT:=UINT_TO_TIME (Ystavki.Yst_Tvkl_AVOM2.Yst_T2 * 1000));
Vkl_AVOM2 (CLK:=(T2_vklAVOM.Q ));
IF	Vkl_AVOM2.Q THEN
	flag_vkl2:=TRUE;
	CASE (num) OF
	4:	IF (num_arr 	[0] =0) THEN
			num:=1;
			num_arr 	[0]:=2;
		END_IF
	0..3:	num_arr 	[num]:= 2;
			num 		:= num + 1;
	END_CASE
	avoms_vkl ();
END_IF
/////////////////////////////////////////////////////////////////////
T3_vklAVOM(IN:=((T_posle_AVOM.interval>=statusAi.NORmaL) AND (T_posle_AVOM.value >= Ystavki.Yst_AVOM_T3.Yst_T3) AND flag_vkl1 AND flag_vkl2 AND NOT flag_vkl3), PT:=UINT_TO_TIME (Ystavki.Yst_Tvkl_AVOM3.Yst_T3 * 1000));
Vkl_AVOM3 (CLK:=(T3_vklAVOM.Q ));
IF	Vkl_AVOM3.Q THEN
	flag_vkl3:=TRUE;
	CASE (num) OF
	4:	IF (num_arr 	[0] =0) THEN
			num:=1;
			num_arr 	[0]:=3;
		END_IF
	0..3:	num_arr 	[num]:= 3;
			num 		:= num + 1;
	END_CASE
	avoms_vkl ();
END_IF
/////////////////////////////////////////////////////////////////////
T4_vklAVOM(IN:=((T_posle_AVOM.interval>=statusAi.NORmaL) AND (T_posle_AVOM.value >= Ystavki.Yst_AVOM_T4.Yst_T4) AND flag_vkl3 AND flag_vkl1 AND flag_vkl2 AND NOT flag_vkl4 ), PT:=UINT_TO_TIME (Ystavki.Yst_Tvkl_AVOM4.Yst_T4 * 1000));
Vkl_AVOM4 (CLK:=(T4_vklAVOM.Q ));
IF	Vkl_AVOM4.Q THEN
	flag_vkl4:=TRUE;
	CASE (num) OF
	4:	IF (num_arr 	[0] =0) THEN
			num:=1;
			num_arr 	[0]:=4;
		END_IF
	0..3:	num_arr 	[num]:= 4;
			num 		:= num + 1;
	END_CASE
	avoms_vkl ();
END_IF
/////////////////////////////////////////////////////////////////////

T1_vyklAVOM(IN:=((T_posle_AVOM.interval>=statusAi.NORmaL) AND (T_posle_AVOM.value <= (Ystavki.Yst_AVOM_T1.Yst_T1 - Ystavki.Yst_DTvykl_AVOM1.Yst_T1)) AND flag_vkl1 AND NOT flag_vkl2), PT:=UINT_TO_TIME (Ystavki.Yst_Tvykl_AVOM1.Yst_T1 * 1000));
Vykl_AVOM1 (CLK:=(T1_vyklAVOM.Q ));
IF	Vykl_AVOM1.Q THEN
	flag_vkl1:=FALSE;
	FOR i:=0 TO 3 DO
		IF 	num_arr [i] > 0 THEN
			num_arr [i] := num_arr [i] - 1;
		END_IF
		IF 	num_arr [i] = 0 THEN
			CASE i OF
				0: num_vykl:= 1;
				1: num_vykl:= 2;
				2: num_vykl:= 3;
				3: num_vykl:= 4;
			END_CASE
			avoms_vykl ();
		END_IF
	END_FOR
	avoms_vykl ();
END_IF
/////////////////////////////////////////////////////////////////////
T2_vyklAVOM(IN:=((T_posle_AVOM.interval>=statusAi.NORmaL) AND (T_posle_AVOM.value <= (Ystavki.Yst_AVOM_T2.Yst_T2 - Ystavki.Yst_DTvykl_AVOM2.Yst_T2)) AND flag_vkl2 AND NOT flag_vkl3), PT:= UINT_TO_TIME (Ystavki.Yst_Tvykl_AVOM2.Yst_T2 * 1000));
Vykl_AVOM2 (CLK:=(T2_vyklAVOM.Q ));
IF	Vykl_AVOM2.Q THEN
	flag_vkl2:=FALSE;
	FOR i:=0 TO 3 DO
		IF 	num_arr [i] > 0 THEN
			num_arr [i] := num_arr [i] - 1;
		END_IF
		IF 	num_arr [i] = 0 THEN
			CASE i OF
				0: num_vykl:= 1;
				1: num_vykl:= 2;
				2: num_vykl:= 3;
				3: num_vykl:= 4;
			END_CASE
			avoms_vykl ();
		END_IF
	END_FOR
	avoms_vykl ();
END_IF
/////////////////////////////////////////////////////////////////////
T3_vyklAVOM(IN:=((T_posle_AVOM.interval>=statusAi.NORmaL) AND (T_posle_AVOM.value <= (Ystavki.Yst_AVOM_T3.Yst_T3 - Ystavki.Yst_DTvykl_AVOM3.Yst_T3)) AND flag_vkl3 AND NOT flag_vkl4), PT:=UINT_TO_TIME (Ystavki.Yst_Tvykl_AVOM3.Yst_T3 * 1000));
Vykl_AVOM3 (CLK:=(T3_vyklAVOM.Q ));
IF	Vykl_AVOM3.Q THEN
	flag_vkl3:=FALSE;
	FOR i:=0 TO 3 DO
		IF 	num_arr [i] > 0 THEN
			num_arr [i] := num_arr [i] - 1;
		END_IF
		IF 	num_arr [i] = 0 THEN
			CASE i OF
				0: num_vykl:= 1;
				1: num_vykl:= 2;
				2: num_vykl:= 3;
				3: num_vykl:= 4;
			END_CASE
			avoms_vykl ();
		END_IF
	END_FOR
	avoms_vykl ();
END_IF
/////////////////////////////////////////////////////////////////////
T4_vyklAVOM(IN:=((T_posle_AVOM.interval>=statusAi.NORmaL) AND (T_posle_AVOM.value <= (Ystavki.Yst_AVOM_T4.Yst_T4 - Ystavki.Yst_DTvykl_AVOM4.Yst_T4)) AND flag_vkl4 ), PT:=UINT_TO_TIME (Ystavki.Yst_Tvykl_AVOM4.Yst_T4 * 1000));
Vykl_AVOM4 (CLK:=(T4_vyklAVOM.Q ));
IF	Vykl_AVOM4.Q THEN
	flag_vkl4:=FALSE;
	FOR i:=0 TO 3 DO
		IF 	num_arr [i] > 0 THEN
			num_arr [i] := num_arr [i] - 1;
		END_IF
		IF 	num_arr [i] = 0 THEN
			CASE i OF
				0: num_vykl:= 1;
				1: num_vykl:= 2;
				2: num_vykl:= 3;
				3: num_vykl:= 4;
			END_CASE
			avoms_vykl ();
		END_IF
	END_FOR
END_IF
/////////////////////////////////////////////////////////////////////
IF	(T_posle_AVOM.interval < statusAi.NORmaL) THEN
	reset ();
END_IF

METHOD PRIVATE AVOMs_Vkl
VAR_INPUT
	
END_VAR
VAR
	
END_VAR
SUPER^();
IF	(Vkl_AVOM1.Q OR Vkl_AVOM2.Q OR Vkl_AVOM3.Q OR Vkl_AVOM4.Q) AND (num <> i1_izm)  AND (num > 0) THEN
	CASE 		Ystavki.num_Avom.Yst [num - 1] OF
		1:		A1.on ();
		2:		A2.on ();
		3:		A3.on ();
		4:		A4.on ();
		
	END_CASE
	
END_IF
i1_izm :=num;
END_METHOD

METHOD PUBLIC reset
VAR_INPUT
END_VAR
SUPER^.reset();
im.v1_Avom.off ();
im.v2_Avom.off ();
im.v3_Avom.off ();
im.v4_Avom.off ();

flag_vkl1:=FALSE;
flag_vkl2:=FALSE;
flag_vkl3:=FALSE;
flag_vkl4:=FALSE;
i:=0;
num_vykl:=0;

num_arr [0]:=0;
num_arr [1]:=0;
num_arr [2]:=0;
num_arr [3]:=0;

i1_izm:=0;
i2_izm:=0;

Num:=0;
	
T1_vklAVOM (IN:=FALSE);
T2_vklAVOM (IN:=FALSE);
T3_vklAVOM (IN:=FALSE);
T4_vklAVOM (IN:=FALSE);
	
T1_vyklAVOM (IN:=FALSE);
T2_vyklAVOM (IN:=FALSE);
T3_vyklAVOM (IN:=FALSE);
T4_vyklAVOM (IN:=FALSE);
	
Vkl_AVOM1 	(clk:=FALSE);
Vkl_AVOM2	(clk:=FALSE);
Vkl_AVOM3	(clk:=FALSE);
Vkl_AVOM4	(clk:=FALSE);
	
Vykl_AVOM1	(clk:=FALSE);
Vykl_AVOM2	(clk:=FALSE);
Vykl_AVOM3	(clk:=FALSE);
Vykl_AVOM4	(clk:=FALSE);
IF	algoritms.F2_Ch.autoAVOM_canrun_flag OR algoritms.F2_R.autoAVOM_canrun_flag THEN
	algoritms.S_AutoAVOM.CanRun:=TRUE;
	algoritms.R_AutoAVom.CanRun:=FALSE;
END_IF
END_METHOD

METHOD PRIVATE AVOMs_Vykl
VAR_INPUT
	
END_VAR
VAR
END_VAR
SUPER^();
IF	(Vykl_AVOM1.Q OR Vykl_AVOM2.Q OR Vykl_AVOM3.Q OR Vykl_AVOM4.Q) AND (num_vykl <> i2_izm)  AND (num_vykl > 0) THEN
	CASE 		Ystavki.num_Avom.Yst [num_vykl - 1] OF
		1:		A1.off ();
		2:		A2.off ();
		3:		A3.off ();
		4:		A4.off ();
	END_CASE
END_IF
i2_izm :=num_vykl;
END_METHOD

METHOD PUBLIC run
VAR_INPUT
END_VAR
SUPER^.run();
algoritms.S_AutoAVOM.CanRun:=FALSE;
algoritms.R_AutoAVom.CanRun:=TRUE;
END_METHOD

END_FUNCTION_BLOCK

// K1/std12k5/nasos/AutoNuAlg_2
	{attribute 'symbol' := 'none'}
FUNCTION_BLOCK AutoNuAlg_2 EXTENDS BaseAlgoritm
VAR_INPUT
	nu:REFERENCE TO NasosNu;
	Di:REFERENCE TO singleSignal;
	di_CK:REFERENCE TO BaseIm;
END_VAR
VAR_OUTPUT
	{attribute 'symbol' := 'read'}
	NU_rez_OFF_Ask:		Question(table:=ADR(ObjectTable)):=			(AnswerVariants:=(Answers.ANS_YES));
	{attribute 'symbol' := 'read'}
	NU_osn_OFF_Ask:		Question(table:=ADR(ObjectTable)):=			(AnswerVariants:=(Answers.ANS_YES));
	flag1:BOOL;
	flag2:BOOL;
	flag3:BOOL;
END_VAR
VAR
	
	pgmLw:TON:=(pt:=T#3S);
	lowPmg:R_TRIG;
	T_vkl_secondNU:TON:=(pt:=T#4S);
	timer_Osn_NU_Off:TON:=(pt:=T#3S);
	
END_VAR


SUPER^();
pgmLw(IN:=(di.Q) OR (ai.PerepadDavlenieMasloGaz.interval>=statusAi.LW));
lowPmg (clk:=pgmLw.Q);
////////////////////Включаем основной насос при давлении меньше 100////////////////////////////
	IF	lowPmg.Q AND NOT (flag1 OR flag2)  THEN
		CASE (im.nu.mainNasos.Value) OF
			0:	im.nu.nu1.on ();
				flag1:=TRUE;
			1:	im.nu.nu2.on ();
				flag2:=TRUE;
		END_CASE
	END_IF
////////////////////Включаем резервный насос при давлении меньше 100////////////////////////////	
	T_vkl_secondNU (In:= ((flag1 OR flag2) AND ((di.Q) OR (ai.PerepadDavlenieMasloGaz.interval>=statusAi.LW)) AND NOT flag3));
	
	IF	T_vkl_secondNU.Q THEN
		IF	flag1 THEN
			im.nu.nu2.on ();
		END_IF
		IF	flag2 THEN
			im.nu.nu1.on ();
		END_IF
		flag3:=TRUE;
	END_IF
////////////////////Отключаем насосы по вопросам диспетчеру или по выдержке 3 сек////////////////////////////

		timer_Osn_NU_Off(In:= ((NOT di.Q) AND ((ai.PerepadDavlenieMasloGaz.interval=statusAi.normal) OR (ai.PerepadDavlenieMasloGaz.interval=statusAi.HL))  AND (di_CK.status = 1) AND (flag1 OR flag2)));
		
		IF	timer_Osn_NU_Off.Q THEN
			NU_osn_OFF_Ask.ask ();
		ELSE
			NU_osn_OFF_Ask.reset ();
		END_IF
		
////////////////////Отключаем основной насос////////////////////////////		
	IF 	(NU_osn_OFF_Ask.answer = Answers.ANS_YES) THEN
		IF 	flag1  THEN
			flag1:=FALSE;
			im.nu.nu1.off (); 
		END_IF
		IF 	flag2 THEN
			flag2:=FALSE;
			im.nu.nu2.off ();	
		END_IF
	END_IF
///////////////////////////////////////////////////////////////////////////////////////////////////////////////////
IF	flag3 AND NOT (flag1 OR flag2) AND (NOT di.Q) AND (di_CK.status = 1) AND ((ai.PerepadDavlenieMasloGaz.interval=statusAi.normal) OR (ai.PerepadDavlenieMasloGaz.interval=statusAi.HL))  THEN
	NU_rez_OFF_Ask.ask ();
ELSE
	NU_rez_OFF_Ask.reset ();	
END_IF
////////////////////Отключаем резервный насос////////////////////////////		
	
	IF	(NU_rez_OFF_Ask.answer = Answers.ANS_YES) THEN
			flag3:=FALSE;
			CASE 	im.nu.mainNasos.Value OF
			0:		im.nu.nu2.off ();
					im.nu.mainNasos.setValue(1);
			1:		im.nu.nu1.off ();
					im.nu.mainNasos.setValue(0);
			END_CASE
		END_IF

METHOD PUBLIC reset
VAR_INPUT
END_VAR
SUPER^.reset();
pgmLw (In:=FALSE);
lowPmg (clk:=FALSE);
NU_rez_OFF_Ask.reset();
NU_osn_OFF_Ask.reset ();
flag1:=FALSE;
flag2:=FALSE;
flag3:=FALSE;
T_vkl_secondNU(In:=FALSE);
timer_Osn_NU_Off (In:=FALSE);
END_METHOD

END_FUNCTION_BLOCK

// K2/std12k5/nasos/AutoNuAlg_2
	{attribute 'symbol' := 'none'}
FUNCTION_BLOCK AutoNuAlg_2 EXTENDS BaseAlgoritm
VAR_INPUT
	nu:REFERENCE TO NasosNu;
	Di:REFERENCE TO singleSignal;
	di_CK:REFERENCE TO BaseIm;
END_VAR
VAR_OUTPUT
	{attribute 'symbol' := 'read'}
	NU_rez_OFF_Ask:		Question(table:=ADR(ObjectTable)):=			(AnswerVariants:=(Answers.ANS_YES));
	{attribute 'symbol' := 'read'}
	NU_osn_OFF_Ask:		Question(table:=ADR(ObjectTable)):=			(AnswerVariants:=(Answers.ANS_YES));
	flag1:BOOL;
	flag2:BOOL;
	flag3:BOOL;
END_VAR
VAR
	
	pgmLw:TON:=(pt:=T#3S);
	lowPmg:R_TRIG;
	T_vkl_secondNU:TON:=(pt:=T#4S);
	timer_Osn_NU_Off:TON:=(pt:=T#3S);
	
END_VAR


SUPER^();
pgmLw(IN:=(di.Q) OR (ai.PerepadDavlenieMasloGaz.interval>=statusAi.LW));
lowPmg (clk:=pgmLw.Q);
////////////////////Включаем основной насос при давлении меньше 100////////////////////////////
	IF	lowPmg.Q AND NOT (flag1 OR flag2)  THEN
		CASE (im.nu.mainNasos.Value) OF
			0:	im.nu.nu1.on ();
				flag1:=TRUE;
			1:	im.nu.nu2.on ();
				flag2:=TRUE;
		END_CASE
	END_IF
////////////////////Включаем резервный насос при давлении меньше 100////////////////////////////	
	T_vkl_secondNU (In:= ((flag1 OR flag2) AND ((di.Q) OR (ai.PerepadDavlenieMasloGaz.interval>=statusAi.LW)) AND NOT flag3));
	
	IF	T_vkl_secondNU.Q THEN
		IF	flag1 THEN
			im.nu.nu2.on ();
		END_IF
		IF	flag2 THEN
			im.nu.nu1.on ();
		END_IF
		flag3:=TRUE;
	END_IF
////////////////////Отключаем насосы по вопросам диспетчеру или по выдержке 3 сек////////////////////////////

		timer_Osn_NU_Off(In:= ((NOT di.Q) AND ((ai.PerepadDavlenieMasloGaz.interval=statusAi.normal) OR (ai.PerepadDavlenieMasloGaz.interval=statusAi.HL))  AND (di_CK.status = 1) AND (flag1 OR flag2)));
		
		IF	timer_Osn_NU_Off.Q THEN
			NU_osn_OFF_Ask.ask ();
		ELSE
			NU_osn_OFF_Ask.reset ();
		END_IF
		
////////////////////Отключаем основной насос////////////////////////////		
	IF 	(NU_osn_OFF_Ask.answer = Answers.ANS_YES) THEN
		IF 	flag1  THEN
			flag1:=FALSE;
			im.nu.nu1.off (); 
		END_IF
		IF 	flag2 THEN
			flag2:=FALSE;
			im.nu.nu2.off ();	
		END_IF
	END_IF
///////////////////////////////////////////////////////////////////////////////////////////////////////////////////
IF	flag3 AND NOT (flag1 OR flag2) AND (NOT di.Q) AND (di_CK.status = 1) AND ((ai.PerepadDavlenieMasloGaz.interval=statusAi.normal) OR (ai.PerepadDavlenieMasloGaz.interval=statusAi.HL))  THEN
	NU_rez_OFF_Ask.ask ();
ELSE
	NU_rez_OFF_Ask.reset ();	
END_IF
////////////////////Отключаем резервный насос////////////////////////////		
	
	IF	(NU_rez_OFF_Ask.answer = Answers.ANS_YES) THEN
			flag3:=FALSE;
			CASE 	im.nu.mainNasos.Value OF
			0:		im.nu.nu2.off ();
					im.nu.mainNasos.setValue(1);
			1:		im.nu.nu1.off ();
					im.nu.mainNasos.setValue(0);
			END_CASE
		END_IF

METHOD PUBLIC reset
VAR_INPUT
END_VAR
SUPER^.reset();
pgmLw (In:=FALSE);
lowPmg (clk:=FALSE);
NU_rez_OFF_Ask.reset();
NU_osn_OFF_Ask.reset ();
flag1:=FALSE;
flag2:=FALSE;
flag3:=FALSE;
T_vkl_secondNU(In:=FALSE);
timer_Osn_NU_Off (In:=FALSE);
END_METHOD

END_FUNCTION_BLOCK

// K2/std12k5/Logic/AI_Final
{attribute 'symbol' := 'none'}
FUNCTION_BLOCK AI_Final EXTENDS AiSourceMlp
VAR_INPUT
	(*n:uint;*)
END_VAR
VAR_OUTPUT
END_VAR
VAR
	
END_VAR

SUPER^();
(*IF	(sip.Yst [n] >=0) AND (sip.Yst [n] <> maxChangeSpeed) THEN
	setNewSIP ();
END_IF*)	IF	dll = STRING_TO_REAL('NaN') THEN
		ll:= dll; 
	END_IF
	IF	dla =STRING_TO_REAL('NaN') THEN
		la:=dla; 
	END_IF
	IF	dlw = STRING_TO_REAL('NaN') THEN	
		lw:=dlw; 
	END_IF
	IF	dhw = STRING_TO_REAL('NaN') THEN
		hw:=dhw; 
	END_IF
	IF	dha = STRING_TO_REAL('NaN') THEN
		ha:=dha; 
	END_IF 
	IF	dhl = STRING_TO_REAL('NaN') THEN
		hl:=dhl; 
	END_IF

METHOD setNewSIP
VAR_INPUT
END_VAR

maxChangeSpeed:=sip.Yst [n];


SaveToFile();
END_METHOD

END_FUNCTION_BLOCK

// K1/std12k5/Logic/AI_Final
{attribute 'symbol' := 'none'}
FUNCTION_BLOCK AI_Final EXTENDS AiSourceMlp
VAR_INPUT
	(*n:uint;*)
END_VAR
VAR_OUTPUT
END_VAR
VAR
	
END_VAR

SUPER^();
	IF	dll = STRING_TO_REAL('NaN') THEN
		ll:= dll; 
	END_IF
	IF	dla =STRING_TO_REAL('NaN') THEN
		la:=dla; 
	END_IF
	IF	dlw = STRING_TO_REAL('NaN') THEN	
		lw:=dlw; 
	END_IF
	IF	dhw = STRING_TO_REAL('NaN') THEN
		hw:=dhw; 
	END_IF
	IF	dha = STRING_TO_REAL('NaN') THEN
		ha:=dha; 
	END_IF 
	IF	dhl = STRING_TO_REAL('NaN') THEN
		hl:=dhl; 
	END_IF

METHOD setNewSIP
VAR_INPUT
END_VAR

maxChangeSpeed:=sip.Yst [n];


SaveToFile();
END_METHOD

END_FUNCTION_BLOCK

// K1/std12k5/nasos/AutoNuAlg_1
	{attribute 'symbol' := 'none'}
FUNCTION_BLOCK AutoNuAlg_1 EXTENDS BaseAlgoritm
VAR_INPUT
	nu:REFERENCE TO NasosNu;
	Di:REFERENCE TO singleSignal;
	di_CK:REFERENCE TO BaseIm ;
END_VAR
VAR_OUTPUT
	{attribute 'symbol' := 'read'}
	NU_OFF_Ask:		Question(table:=ADR(ObjectTable)):=			(AnswerVariants:=(Answers.ANS_YES));
	flag1:BOOL;
	flag2:BOOL;

END_VAR
VAR
	change_NU:WORD;
	pgmLw:TON:=(pt:=T#3S);
	lowPmg:R_TRIG;
	timer3_Sec:TON:=(pt:=T#3S);
	
END_VAR


SUPER^();
pgmLw(IN:=(di.Q) OR (ai.PerepadDavlenieMasloGaz.interval>=statusAi.LW));
lowPmg (clk:=pgmLw.Q);
///////////Выбор НУ при давлении больше 100/////////////////////////////////////

	IF	(NOT di.Q) AND (di_CK.status = 1) AND NOT (flag1 OR flag2) AND (change_NU <> im.nu.mainNasos.Value) AND ((ai.PerepadDavlenieMasloGaz.interval=statusAi.normal)
		OR (ai.PerepadDavlenieMasloGaz.interval=statusAi.HL)) THEN
		CASE	(im.nu.mainNasos.Value) OF
		0:		im.nu.nu1.on ();
				im.nu.nu2.off ();
		1:		im.nu.nu1.off ();
				im.nu.nu2.on ();
		END_CASE
	END_IF
	change_NU := im.nu.mainNasos.Value;
///////////Включаем резервный насос при давлении меньше 100/////////////////////////////////////
	IF	lowPmg.Q AND NOT (flag1 OR flag2) THEN
		CASE	(im.nu.mainNasos.Value) OF
			0:	im.nu.nu2.on ();
				flag1:=TRUE;
			1:	im.nu.nu1.on ();
				flag2:=TRUE;
		END_CASE
	END_IF
///////////После выдержки 3 сек или по команде оператора отключаем насосы/////////////////////////////////////

		timer3_Sec(IN:=	((flag1 OR flag2) AND (NOT di.Q) AND (di_CK.status = 1) AND ((ai.PerepadDavlenieMasloGaz.interval=statusAi.normal) OR (ai.PerepadDavlenieMasloGaz.interval=statusAi.HL))));
	
		IF	timer3_Sec.Q  THEN
			NU_OFF_Ask.ask ();
		ELSE	
			NU_OFF_Ask.reset ();
		END_IF
		
///////////После выдержки 3 сек или по команде оператора отключаем насосы/////////////////////////////////////	
	IF	(NU_OFF_Ask.answer = Answers.ANS_YES) THEN
		IF 	flag1 THEN
			flag1:=FALSE;
			im.nu.nu1.off ();
			im.nu.mainNasos.setvalue (1);
		END_IF
		IF 	flag2  THEN
			flag2:=FALSE;
			im.nu.nu2.off ();
			im.nu.mainNasos.setvalue (0);
		END_IF
	END_IF

METHOD PUBLIC reset
VAR_INPUT
END_VAR
SUPER^.reset();
pgmLw (In:=FALSE);
lowPmg (clk:=FALSE);
NU_OFF_Ask.reset ();
flag1:=FALSE;
flag2:=FALSE;

change_NU:=0;
timer3_Sec(In:=FALSE);
END_METHOD

END_FUNCTION_BLOCK

// K2/std12k5/nasos/AutoNuAlg_1
	{attribute 'symbol' := 'none'}
FUNCTION_BLOCK AutoNuAlg_1 EXTENDS BaseAlgoritm
VAR_INPUT
	nu:REFERENCE TO NasosNu;
	Di:REFERENCE TO singleSignal;
	di_CK:REFERENCE TO BaseIm ;
END_VAR
VAR_OUTPUT
	{attribute 'symbol' := 'read'}
	NU_OFF_Ask:		Question(table:=ADR(ObjectTable)):=			(AnswerVariants:=(Answers.ANS_YES));
	flag1:BOOL;
	flag2:BOOL;

END_VAR
VAR
	change_NU:WORD;
	pgmLw:TON:=(pt:=T#3S);
	lowPmg:R_TRIG;
	timer3_Sec:TON:=(pt:=T#3S);
	
END_VAR


SUPER^();
pgmLw(IN:=(di.Q) OR (ai.PerepadDavlenieMasloGaz.interval>=statusAi.LW));
lowPmg (clk:=pgmLw.Q);
///////////Выбор НУ при давлении больше 100/////////////////////////////////////

	IF	(NOT di.Q) AND (di_CK.status = 1) AND NOT (flag1 OR flag2) AND (change_NU <> im.nu.mainNasos.Value) AND ((ai.PerepadDavlenieMasloGaz.interval=statusAi.normal)
		OR (ai.PerepadDavlenieMasloGaz.interval=statusAi.HL)) THEN
		CASE	(im.nu.mainNasos.Value) OF
		0:		im.nu.nu1.on ();
				im.nu.nu2.off ();
		1:		im.nu.nu1.off ();
				im.nu.nu2.on ();
		END_CASE
	END_IF
	change_NU := im.nu.mainNasos.Value;
///////////Включаем резервный насос при давлении меньше 100/////////////////////////////////////
	IF	lowPmg.Q AND NOT (flag1 OR flag2) THEN
		CASE	(im.nu.mainNasos.Value) OF
			0:	im.nu.nu2.on ();
				flag1:=TRUE;
			1:	im.nu.nu1.on ();
				flag2:=TRUE;
		END_CASE
	END_IF
///////////После выдержки 3 сек или по команде оператора отключаем насосы/////////////////////////////////////

		timer3_Sec(IN:=	((flag1 OR flag2) AND (NOT di.Q) AND (di_CK.status = 1) AND ((ai.PerepadDavlenieMasloGaz.interval=statusAi.normal) OR (ai.PerepadDavlenieMasloGaz.interval=statusAi.HL))));
	
		IF	timer3_Sec.Q  THEN
			NU_OFF_Ask.ask ();
		ELSE	
			NU_OFF_Ask.reset ();
		END_IF
		
///////////После выдержки 3 сек или по команде оператора отключаем насосы/////////////////////////////////////	
	IF	(NU_OFF_Ask.answer = Answers.ANS_YES) THEN
		IF 	flag1 THEN
			flag1:=FALSE;
			im.nu.nu1.off ();
			im.nu.mainNasos.setvalue (1);
		END_IF
		IF 	flag2  THEN
			flag2:=FALSE;
			im.nu.nu2.off ();
			im.nu.mainNasos.setvalue (0);
		END_IF
	END_IF

METHOD PUBLIC reset
VAR_INPUT
END_VAR
SUPER^.reset();
pgmLw (In:=FALSE);
lowPmg (clk:=FALSE);
NU_OFF_Ask.reset ();
flag1:=FALSE;
flag2:=FALSE;

change_NU:=0;
timer3_Sec(In:=FALSE);
END_METHOD

END_FUNCTION_BLOCK

// K1/std12k5/nasos/AutoPnsALg
	{attribute 'symbol' := 'none'}
FUNCTION_BLOCK AutoPnsALg EXTENDS BaseAlgoritm
VAR_INPUT
	Psm_GNS :REFERENCE TO AiSource;
	pns:REFERENCE TO Nasos;
	{attribute 'symbol' := 'read'}
	Auto:DiscretParametr(table:=ADR(objectTable));//{name:режим работы защиты}
END_VAR
VAR_OUTPUT
	{attribute 'symbol' := 'read'}
	PNS_Off:	Question(table:=ADR(ObjectTable)):=			(AnswerVariants:=(Answers.ANS_YES ));
	PNS_OFF_Timer:TON:=(pt:=T#30S);
	{attribute 'symbol' := 'read'}
	Timer_PNS_Off30:REAL;
END_VAR
VAR
	Psm_niz:BOOL;
	Psm_vis:BOOL;
	psmLw:TON:=(pt:=T#4S);
	psmHw:TON:=(pt:=T#4S);
	psmLwTrig:R_TRIG;
	psmHwTrig:R_TRIG;
	flag1:BOOL;
	
END_VAR

SUPER^();
IF	((Psm_GNS.interval>=statusAi.NORMAL) AND (Psm_GNS.AiValue < Ystavki.YstPNS_YP.Yst)) THEN
	Psm_niz := TRUE;
ELSE
	Psm_niz := FALSE;
END_IF
////////////////////////////////
psmLw(IN:=Psm_niz);
psmLwTrig (CLk:=psmLw.Q);
////////////////////////////////
IF	psmLwTrig.Q AND NOT flag1 THEN
	pns.on();	
	flag1:=TRUE;
	
END_IF
////////////////////////////////
IF	((Psm_GNS.interval>=statusAi.NORMAL) AND (Psm_GNS.AiValue > Ystavki.YstPNS_YT.Yst)) AND flag1 THEN
	Psm_vis := TRUE;
ELSE
	Psm_vis := FALSE;
END_IF
psmHw(IN:=Psm_vis);


IF	(Auto.value = 0)	 THEN
	PNS_OFF_Timer (IN:=psmHw.Q);
	Timer_PNS_Off30:=(30 - (TIME_TO_REAL (PNS_OFF_Timer.ET)/1000));
	psmHwTrig (CLk:=PNS_OFF_Timer.Q);
	IF	psmHwTrig.Q THEN
		pns.off();
		
		flag1:=FALSE;
	END_IF
	PNS_Off.reset ();
ELSE
	Timer_PNS_Off30:=30;
	PNS_OFF_Timer (in:=FALSE);
	psmHwTrig(clk:=FALSE);
	IF	psmHw.Q THEN
		PNS_Off.ask ();
	ELSE
		PNS_Off.reset ();
	END_IF
	IF	PNS_Off.answer=Answers.ANS_YES THEN
		pns.off();
		
		flag1:=FALSE;
		PNS_Off.reset ();
	END_IF
END_IF

METHOD PUBLIC reset
VAR_INPUT
END_VAR
SUPER^.reset();
PNS_Off.reset ();
PNS_OFF_Timer(in:=FALSE);
Timer_PNS_Off30:=0;
Psm_niz:=FALSE;
Psm_vis:=FALSE;
psmLw(IN:=FALSE);
psmHw(IN:=FALSE);
psmLwTrig(clk:=FALSE);
psmHwTrig(clk:=FALSE);
flag1:=FALSE;
END_METHOD

END_FUNCTION_BLOCK

// K2/std12k5/nasos/AutoPnsALg
	{attribute 'symbol' := 'none'}
FUNCTION_BLOCK AutoPnsALg EXTENDS BaseAlgoritm
VAR_INPUT
	Psm_GNS :REFERENCE TO AiSource;
	pns:REFERENCE TO Nasos;
	{attribute 'symbol' := 'read'}
	Auto:DiscretParametr(table:=ADR(objectTable));//{name:режим работы защиты}
END_VAR
VAR_OUTPUT
	{attribute 'symbol' := 'read'}
	PNS_Off:	Question(table:=ADR(ObjectTable)):=			(AnswerVariants:=(Answers.ANS_YES ));
	PNS_OFF_Timer:TON:=(pt:=T#30S);
	{attribute 'symbol' := 'read'}
	Timer_PNS_Off30:REAL;
END_VAR
VAR
	Psm_niz:BOOL;
	Psm_vis:BOOL;
	psmLw:TON:=(pt:=T#4S);
	psmHw:TON:=(pt:=T#4S);
	psmLwTrig:R_TRIG;
	psmHwTrig:R_TRIG;
	flag1:BOOL;
	
END_VAR

SUPER^();
IF	((Psm_GNS.interval>=statusAi.NORMAL) AND (Psm_GNS.AiValue < Ystavki.YstPNS_YP.yst)) THEN
	Psm_niz := TRUE;
ELSE
	Psm_niz := FALSE;
END_IF
////////////////////////////////
psmLw(IN:=Psm_niz);
psmLwTrig (CLk:=psmLw.Q);
////////////////////////////////
IF	psmLwTrig.Q AND NOT flag1 THEN
	pns.on();	
	flag1:=TRUE;
	
END_IF
////////////////////////////////
IF	((Psm_GNS.interval>=statusAi.NORMAL) AND (Psm_GNS.AiValue > Ystavki.YstPNS_YT.yst)) AND flag1 THEN
	Psm_vis := TRUE;
ELSE
	Psm_vis := FALSE;
END_IF
psmHw(IN:=Psm_vis);


IF	(Auto.value = 0)	 THEN
	PNS_OFF_Timer (IN:=psmHw.Q);
	Timer_PNS_Off30:=(30 - (TIME_TO_REAL (PNS_OFF_Timer.ET)/1000));
	psmHwTrig (CLk:=PNS_OFF_Timer.Q);
	IF	psmHwTrig.Q THEN
		pns.off();
		
		flag1:=FALSE;
	END_IF
	PNS_Off.reset ();
ELSE
	Timer_PNS_Off30:=30;
	PNS_OFF_Timer (in:=FALSE);
	psmHwTrig(clk:=FALSE);
	IF	psmHw.Q THEN
		PNS_Off.ask ();
	ELSE
		PNS_Off.reset ();
	END_IF
	IF	PNS_Off.answer=Answers.ANS_YES THEN
		pns.off();
		
		flag1:=FALSE;
		PNS_Off.reset ();
	END_IF
END_IF

METHOD PUBLIC reset
VAR_INPUT
END_VAR
SUPER^.reset();
PNS_Off.reset ();
PNS_OFF_Timer(in:=FALSE);
Timer_PNS_Off30:=0;
Psm_niz:=FALSE;
Psm_vis:=FALSE;
psmLw(IN:=FALSE);
psmHw(IN:=FALSE);
psmLwTrig(clk:=FALSE);
psmHwTrig(clk:=FALSE);
flag1:=FALSE;
END_METHOD

END_FUNCTION_BLOCK

// K1/std12k5/nasos/AutoTEN
	{attribute 'symbol' := 'none'}
FUNCTION_BLOCK AutoTEN EXTENDS BaseAlgoritm
VAR_INPUT
	TEN:REFERENCE TO Nasos;
	CMN:REFERENCE TO Nasos;
	Tmb:REFERENCE TO AiSource;
	TmbTEN:REFERENCE TO AiSource;
END_VAR
VAR_OUTPUT
END_VAR
VAR
	TLw:TON:=(pt:=T#3S);
	THw:TON:=(pt:=T#3S);
	TmbLwTrig:R_TRIG;
	TmbHwTrig:R_TRIG;
	flag1:BOOL;
	flag2:BOOL;
	Reset_alg:BOOL;
END_VAR

SUPER^();
Reset_alg:= ((cmn.onStatus <> statusDualInput.status_on)  AND (ten.onStatus = statusDualInput.status_on)) OR 
			(Tmb.interval < statusAi.Normal) OR (TmbTEN.interval = statusAi.HW) OR (TmbTEN.interval < statusAi.Normal) OR (ai.YrovenMaslaMB.interval <> statusAi.Normal);
			
TLw(IN:=((Tmb.interval>=statusAi.Normal) AND (Tmb.value < Ystavki.Yst_Vkl_TEN.Yst_vkl_TEN) AND NOT Reset_alg));
TmbLwTrig(CLK:=TLw.Q);

IF	TmbLwTrig.Q AND NOT flag1 AND NOT Reset_alg  THEN	
	CMN.on(); 
	flag1:=TRUE;
	flag2:=FALSE;
END_IF

IF	(CMN.onStatus = statusDualInput.status_on) AND flag1 AND NOT Reset_alg THEN
	TEN.on ();
END_IF

THw(IN:=((Tmb.interval>=statusAi.Normal) AND (Tmb.value > Ystavki.Yst_Vykl_TEN.Yst_vykl_TEN)));
TmbHwTrig(CLK:=THw.Q);

IF	TmbHwTrig.Q AND NOT flag2 THEN
	TEN.off();
	flag1:=FALSE;
	flag2:=TRUE;
END_IF

IF	TEN.onStatus = statusDualInput.status_off AND flag2 THEN
	CMN.off ();
END_IF
(*
IF	(cmn.onStatus <> statusDualInput.status_on)  AND (ten.onStatus = statusDualInput.status_on) THEN
	CMN.off ();
END_IF
*)
IF	(*(Tmb.interval < statusAi.Normal) OR (TmbTEN.interval >= statusAi.LW)*) Reset_alg THEN
	reset ();
END_IF

METHOD PUBLIC run
VAR_INPUT
END_VAR
SUPER^.run();
algoritms.S_AutoTEN.CanRun:=FALSE;
algoritms.R_AutoTEN.CanRun:=TRUE;
END_METHOD

METHOD PUBLIC reset
VAR_INPUT
END_VAR
SUPER^.reset();
im.TEN_MB.off ();
im.CMN.off ();
TLw(IN:=FALSE);
THw(IN:=FALSE);
TmbLwTrig(clk:=FALSE);
TmbHwTrig(clk:=FALSE);
flag1:=FALSE;
flag2:=FALSE;
IF	(algmanager.mode=modegpa.MODE_STOP) THEN
	algoritms.S_AutoTEN.CanRun:=TRUE;
	algoritms.R_AutoTEN.CanRun:=FALSE;
END_IF
END_METHOD

END_FUNCTION_BLOCK

// lowLevel_ecl/im/ventvs/Ten
	{attribute 'symbol' := 'none'}
FUNCTION_BLOCK Ten EXTENDS Ventvs
VAR_INPUT
END_VAR
VAR_OUTPUT
END_VAR
VAR
END_VAR

SUPER^();

END_FUNCTION_BLOCK

// K2/std12k5/nasos/AutoTEN
	{attribute 'symbol' := 'none'}
FUNCTION_BLOCK AutoTEN EXTENDS BaseAlgoritm
VAR_INPUT
	TEN:REFERENCE TO Nasos;
	CMN:REFERENCE TO Nasos;
	Tmb:REFERENCE TO AiSource;
	TmbTEN:REFERENCE TO AiSource;
END_VAR
VAR_OUTPUT
END_VAR
VAR
	TLw:TON:=(pt:=T#3S);
	THw:TON:=(pt:=T#3S);
	TmbLwTrig:R_TRIG;
	TmbHwTrig:R_TRIG;
	flag1:BOOL;
	flag2:BOOL;
	Reset_alg:BOOL;
END_VAR

SUPER^();
Reset_alg:= ((cmn.onStatus <> statusDualInput.status_on)  AND (ten.onStatus = statusDualInput.status_on)) OR 
			(Tmb.interval < statusAi.Normal) OR (TmbTEN.interval = statusAi.HW) OR (TmbTEN.interval < statusAi.Normal) OR (ai.YrovenMaslaMB.interval <> statusAi.Normal);
			
TLw(IN:=((Tmb.interval>=statusAi.Normal) AND (Tmb.value < Ystavki.Yst_Vkl_TEN.Yst_vkl_TEN) AND NOT Reset_alg));
TmbLwTrig(CLK:=TLw.Q);

IF	TmbLwTrig.Q AND NOT flag1 AND NOT Reset_alg  THEN	
	CMN.on(); 
	flag1:=TRUE;
	flag2:=FALSE;
END_IF

IF	(CMN.onStatus = statusDualInput.status_on) AND flag1 AND NOT Reset_alg THEN
	TEN.on ();
END_IF

THw(IN:=((Tmb.interval>=statusAi.Normal) AND (Tmb.value > Ystavki.Yst_Vykl_TEN.Yst_vykl_TEN)));
TmbHwTrig(CLK:=THw.Q);

IF	TmbHwTrig.Q AND NOT flag2 THEN
	TEN.off();
	flag1:=FALSE;
	flag2:=TRUE;
END_IF

IF	TEN.onStatus = statusDualInput.status_off AND flag2 THEN
	CMN.off ();
END_IF
(*
IF	(cmn.onStatus <> statusDualInput.status_on)  AND (ten.onStatus = statusDualInput.status_on) THEN
	CMN.off ();
END_IF
*)
IF	(*(Tmb.interval < statusAi.Normal) OR (TmbTEN.interval >= statusAi.LW)*) Reset_alg THEN
	reset ();
END_IF

METHOD PUBLIC run
VAR_INPUT
END_VAR
SUPER^.run();
algoritms.S_AutoTEN.CanRun:=FALSE;
algoritms.R_AutoTEN.CanRun:=TRUE;
END_METHOD

METHOD PUBLIC reset
VAR_INPUT
END_VAR
SUPER^.reset();
im.TEN_MB.off ();
im.CMN.off ();
TLw(IN:=FALSE);
THw(IN:=FALSE);
TmbLwTrig(clk:=FALSE);
TmbHwTrig(clk:=FALSE);
flag1:=FALSE;
flag2:=FALSE;
IF	(algmanager.mode=modegpa.MODE_STOP) THEN
	algoritms.S_AutoTEN.CanRun:=TRUE;
	algoritms.R_AutoTEN.CanRun:=FALSE;
END_IF
END_METHOD

END_FUNCTION_BLOCK

// K1/std12k5/nasos/PNS_ON_MV_ON
{attribute 'symbol' := 'none'}
FUNCTION_BLOCK PNS_ON_MV_ON EXTENDS BaseAlgoritm
VAR_INPUT
	PNS:REFERENCE TO Nasos;
END_VAR
VAR_OUTPUT
END_VAR
VAR
	TPNS:TON:=(pt:=T#3S);
	PNS_On:R_TRIG;
END_VAR

SUPER^();
TPNS (IN:= (im.mv.onStatus=statusDualInput.status_on));
PNS_On (clk:=TPNS.Q);
IF	PNS_On.Q THEN
	PNS.on();
END_IF

METHOD PUBLIC reset
VAR_INPUT
END_VAR
SUPER^.reset();
TPNS(in:=FALSE);
PNS_On(clk:=FALSE);
END_METHOD

END_FUNCTION_BLOCK

// K2/std12k5/nasos/PNS_ON_MV_ON
{attribute 'symbol' := 'none'}
FUNCTION_BLOCK PNS_ON_MV_ON EXTENDS BaseAlgoritm
VAR_INPUT
	PNS:REFERENCE TO Nasos;
END_VAR
VAR_OUTPUT
END_VAR
VAR
	TPNS:TON:=(pt:=T#3S);
	PNS_On:R_TRIG;
END_VAR

SUPER^();
TPNS (IN:= (im.mv.onStatus=statusDualInput.status_on));
PNS_On (clk:=TPNS.Q);
IF	PNS_On.Q THEN
	PNS.on();
END_IF

METHOD PUBLIC reset
VAR_INPUT
END_VAR
SUPER^.reset();
TPNS(in:=FALSE);
PNS_On(clk:=FALSE);
END_METHOD

END_FUNCTION_BLOCK

// K1/std12k5/OpcCommands
	{attribute 'symbol' := 'none'}
FUNCTION_BLOCK OpcCommands EXTENDS baseAlgoritm
VAR_INPUT
END_VAR
VAR_OUTPUT
END_VAR
VAR
END_VAR

ExecKontrollersComands(table:=kontrollers);

ExecComands(imTable);

algManager.execCommand();
protectmanager.execCommand();
ExecComands(YstTable);

END_FUNCTION_BLOCK

// K2/std12k5/OpcCommands
	{attribute 'symbol' := 'none'}
FUNCTION_BLOCK OpcCommands EXTENDS baseAlgoritm
VAR_INPUT
END_VAR
VAR_OUTPUT
END_VAR
VAR
END_VAR

ExecKontrollersComands(table:=kontrollers);

ExecComands(imTable);

algManager.execCommand();
protectmanager.execCommand();
ExecComands(YstTable);

END_FUNCTION_BLOCK

// K1/std12k5/ostanov/aoAlg
	{attribute 'symbol' := 'none'}
FUNCTION_BLOCK aoAlg EXTENDS StepBySteapAlgoritm
VAR_INPUT
END_VAR
VAR_OUTPUT
	{attribute 'symbol' := 'read'}
	sbrosVibeg:		Question(table:=ADR(ObjectTable)):=			(AnswerVariants:=Answers.ANS_YES);
END_VAR
VAR
	
	kran6Open:		ph_Kran (table:=ADR(phasesTable)):=				(phaseNumber:=0, Im:=Im.kran6, act:=DualStateImAction.on);
	
	kran4Close:		ph_Kran (table:=ADR(phasesTable)):=				(phaseNumber:=1, Im:=Im.kran4, act:=DualStateImAction.off);
	
	kran3bOpen:		ph_Kran (table:=ADR(phasesTable)):=				(phaseNumber:=2, Im:=Im.kran3b, act:=DualStateImAction.on);
	
	mvOff:			ph_Switch (table:=ADR(phasesTable)):=			(phaseNumber:=3, Im:=Im.mv, act:=DualStateImAction.off);
	
	kran1Close:		ph_Kran (table:=ADR(phasesTable)):=				(phaseNumber:=4, Im:=Im.kran1, act:=DualStateImAction.off);
	
	kran2Close:		ph_Kran (table:=ADR(phasesTable)):=				(phaseNumber:=5, Im:=Im.kran2, act:=DualStateImAction.off);
	
	kran3Close:		ph_Kran (table:=ADR(phasesTable)):=				(phaseNumber:=6, Im:=Im.kran3, act:=DualStateImAction.off);
	
	kran5Open:		ph_Kran (table:=ADR(phasesTable)):=				(phaseNumber:=7, Im:=Im.kran5, act:=DualStateImAction.on);
	
	autoPnsOff:		ph_algoritm (table:=ADR(phasesTable)):=			(phaseNumber:=8, Im:=algoritms.autoPns, act:=PhaseAlgoritmAction.reset, waitCompletion:=FALSE);
	
	pnsOn:			ph_Switch (table:=ADR(phasesTable)):=			(phaseNumber:=9, Im:=Im.pns, act:=DualStateImAction.on);
	
	Pg_VhodLessThen300:	CustomPhase (table:=ADR(phasesTable)):=		(phaseNumber:=10);
	
	Pg_VyhodLessThen300:CustomPhase (table:=ADR(phasesTable)):=		(phaseNumber:=11);
	
	nuOff:			ph_Switch (table:=ADR(phasesTable)):=			(phaseNumber:=12, Im:=Im.nu, act:=DualStateImAction.off);
	Auto_NU_Off:	CustomPhase (table:=ADR(phasesTable)):=		(phaseNumber:=13);
	{attribute 'symbol' := 'read'}
	timer600:		ph_Timer (table:=ADR(phasesTable)):=			(phaseNumber:=14, delay:=T#600S);
	
	pnsOff:			ph_Switch (table:=ADR(phasesTable)):=			(phaseNumber:=15, Im:=Im.pns, act:=DualStateImAction.off);
	
	Avom1Off:		ph_Switch (table:=ADR(phasesTable)):=			(phaseNumber:=16, Im:=Im.v1_Avom, act:=DualStateImAction.off);
	
	Avom2Off:		ph_Switch (table:=ADR(phasesTable)):=			(phaseNumber:=17, Im:=Im.v2_Avom, act:=DualStateImAction.off);
	
	Avom3Off:		ph_Switch (table:=ADR(phasesTable)):=			(phaseNumber:=18, Im:=Im.v3_Avom, act:=DualStateImAction.off);
	
	Avom4Off:		ph_Switch (table:=ADR(phasesTable)):=			(phaseNumber:=19, Im:=Im.v4_Avom, act:=DualStateImAction.off);
	
	autoAVOMOff:	ph_algoritm (table:=ADR(phasesTable)):=			(phaseNumber:=20, Im:=algoritms.Auto_Avom_, act:=PhaseAlgoritmAction.reset, waitCompletion:=FALSE);
	
	timer5:			ph_Timer (table:=ADR(phasesTable)):=			(phaseNumber:=21, delay:=T#5S);
	
	klapan1:		CustomPhase (table:=ADR(phasesTable)):=			(phaseNumber:=22);
	
	klapan2:		CustomPhase (table:=ADR(phasesTable)):=			(phaseNumber:=23);
	
	nu_On:			CustomPhase (table:=ADR(phasesTable)):=			(phaseNumber:=24);
	flag1:BOOL;
	Start_AO_From:			CustomPhase (table:=ADR(phasesTable)):=			(phaseNumber:=25);
END_VAR

SUPER^();

//////////////Старт смазки кранов 1 и 2///////////////////////////
IF	algoritms.F3.Smazka_1_2 OR (im.kran1.onStatus = statusDualInput.STATUS_ON) OR (im.kran1.onStatus = statusDualInput.STATUS_TRANSITIONAL)
	OR (im.kran2.onStatus = statusDualInput.STATUS_ON) OR (im.kran2.onStatus = statusDualInput.STATUS_TRANSITIONAL)  THEN
	IF	(algoritms.F3.Smazka_1_2 OR (im.kran1.onStatus = statusDualInput.STATUS_ON) OR (im.kran1.onStatus = statusDualInput.STATUS_TRANSITIONAL)) AND (NOT klapan1.start) AND (NOT kran1Close.top) THEN
		klapan1.run ();
	END_IF
	IF	(algoritms.F3.Smazka_1_2 OR (im.kran2.onStatus = statusDualInput.STATUS_ON) OR (im.kran2.onStatus = statusDualInput.STATUS_TRANSITIONAL)) AND (NOT klapan2.start) AND (NOT kran2Close.top) THEN
		klapan2.run ();
	END_IF
	algoritms.F3.Smazka_1_2:=FALSE;
END_IF

//////////////Переставляем краны///////////////////////////
IF	NOT kran6Open.start THEN
	ystavki.Block_kr6_alg.setValue (1);
	IF	im.kran6._cmdreset.IN = FALSE THEN
		ystavki.Block_kr6_alg.setValue (0);
		kran6Open.run(); //открываем карн 6
	END_IF
END_IF

IF	NOT kran4Close.start THEN
	ystavki.Block_kr4_alg.setValue (1);
	IF	im.kran4._cmdreset.IN = FALSE THEN
		ystavki.Block_kr4_alg.setValue (0);
		kran4Close.run(); //закрываем кран 4
	END_IF
END_IF

IF	NOT kran3bOpen.start THEN
	ystavki.Block_kr3b_alg.setValue (1);
	IF	im.kran3b._cmdreset.IN = FALSE THEN
		ystavki.Block_kr3b_alg.setValue (0);
		kran3bOpen.run (); //Открываем кран 3бис
	END_IF
END_IF
protections.p_mvOff.reset ();
protections.p_OFFAvarSwitch.reset();
protections.p_RegVozbOff.reset ();
protections.p_kran1.reset ();
protections.p_kran2.reset ();
mvOff.run(); //отключаем МВ

IF	NOT kran1Close.start THEN
	ystavki.Block_kr1_alg.setValue (1);
	IF	im.kran1._cmdreset.IN = FALSE THEN
		ystavki.Block_kr1_alg.setValue (0);
		kran1Close.run(); //закрываем кран 1
	END_IF
END_IF

IF	NOT	kran2Close.start THEN
	ystavki.Block_kr2_alg.setValue (1);
	IF	im.kran2._cmdreset.IN = FALSE THEN
		ystavki.Block_kr2_alg.setValue (0);
		kran2Close.run(); //закрываем кран 2 
	END_IF
END_IF

IF	NOT	kran3Close.start THEN
	ystavki.Block_kr3_alg.setValue (1);
	IF	im.kran3._cmdreset.IN = FALSE THEN
		ystavki.Block_kr3_alg.setValue (0);
		kran3Close.run(); //закрываем кран 3
	END_IF
END_IF

IF	kran6Open.top THEN
	algoritms.S_Vibr.CanRun:=FALSE;
	algoritms.S_Vibr.reset ();
END_IF
///////////////выдаем смазку кранов 1 и 2//////////////////////////
IF	klapan1.start AND kran1Close.top THEN
	im.Kr1_Smazka.impulse();//выдача команды на клапан
	klapan1.top:=TRUE;
END_IF;
IF	klapan2.start AND kran2Close.top THEN
	im.Kr2_Smazka.impulse();//выдача команды на клапан
	klapan2.top:=TRUE;
END_IF;
///////////////открываем кран 5//////////////////////////
IF 	kran1Close.top AND kran2Close.top AND kran3Close.top AND kran4Close.top AND NOT kran5Open.top THEN //если кран 1 и 2 закрыты открываем кран 5
	IF	NOT	kran5Open.start THEN
		ystavki.Block_kr5_alg.setValue (1);
		IF	im.kran5._cmdreset.IN = FALSE THEN
			ystavki.Block_kr5_alg.setValue (0);
			kran5Open.run();
		END_IF
	END_IF

	//protections.p_DGazaNaVhodeNagnetatelja.reset ();
	protections.p_DGazaNaVyhodeNagnetatelja.reset ();
END_IF 
/////////////////////////////////////////
IF	mvOff.top AND NOT flag1 THEN //если МВ отключился 
	algoritms.AutoPNS_Start.canrun :=FALSE;
	algoritms.AutoPNS_Start.reset ();
	algoritms.autoPns.canrun :=FALSE;
	autoPnsOff.run ();
	pnsOn.run ();
	nu_On.run();
	CASE 	im.nu.mainNasos.Value OF
	0:		im.nu.nu1.on ();
	1:		im.nu.nu2.on ();
	END_CASE
	algoritms.autoNu_2.canrun:=FALSE;
	algoritms.autoNu_2.reset ();
	algoritms.autoNu_1.canrun:=TRUE;
	algoritms.autoNu_1.run ();
	flag1:=TRUE;
END_IF
IF	((im.nu.nu1.onStatus =statusDualInput.STATUS_On) OR (im.nu.nu2.onStatus =statusDualInput.STATUS_On)) AND nu_On.start AND NOT nu_On.top THEN
	nu_On.top:=TRUE;
END_IF
/////////////////////////////////////////
IF 	kran5Open.top THEN //если отключены МВ и 5 кран
	Pg_VhodLessThen300.run();  //проверяем условие, что давление в нагнетателе меньше 100
	Pg_VyhodLessThen300.run(); 
	
END_IF 
/////////////////////////////////////////
IF Pg_VhodLessThen300.start AND (NOT Pg_VhodLessThen300.top) THEN
	IF 	(ai.DGazaNaVhodeNagnetatelja.interval>=statusAi.NORMAL) AND (ai.DGazaNaVhodeNagnetatelja.value < 0.3 )THEN
		Pg_VhodLessThen300.top:=TRUE; //давление в полости нагнетателя меньше 100 кПа
	END_IF
END_IF
/////////////////////////////////////////
IF Pg_VyhodLessThen300.start AND (NOT Pg_VyhodLessThen300.top) THEN
	IF 	(ai.DGazaNaVyhodeNagnetatelja.interval>=statusAi.NORMAL) AND (ai.DGazaNaVyhodeNagnetatelja.value < 0.3) THEN
		Pg_VyhodLessThen300.top:=TRUE; //давление в полости нагнетателя меньше 100 кПа
	END_IF
END_IF
/////////////////////////////////////////
IF 	Pg_VhodLessThen300.top AND Pg_VyhodLessThen300.top AND pnsOn.top AND nu_On.top AND mvOff.top THEN //давление меньше 100 и кран5 и пнс включен 
	nuOff.run(); //отключаем НУ
	protections.p_PerepadDavlenieMasloGaz.reset();
	protections.p_PerepadDavlenieMasloGaz_Less100.reset();
	
	protections.p_DGazaNaVhodeNagnetatelja_GPA_STOP.run ();
	protections.p_DGazaNaVyhodeNagnetatelja_GPA_STOP.run ();
	Auto_NU_Off.top:=TRUE;
	algoritms.autoNu_1.CanRun:=FALSE;
	algoritms.autoNu_1.reset ();
END_IF
/////////////////////////////////////////
IF	nuOff.top THEN //при отключенном ну можо сбросить выбег
	IF	NOT algmanager.reg_V AND NOT pnsoff.start THEN
		timer600.run();
	END_IF;
	IF	NOT pnsoff.start THEN
		sbrosVibeg.ask();
	END_IF;
END_IF
/////////////////////////////////////////
IF 	((timer600.top) OR (sbrosVibeg.answer=Answers.ANS_YES))   THEN //Если прошло 480 секунд и НУ выключен или нажата сброс выбега
	pnsOff.run();//отключаем ПНС
	protections.p_DavlenijaMasloSmNizkoe.reset ();
	protections.p_DavlenijaMasloSmVysokoe.reset ();
	sbrosVibeg.reset ();
	timer600.reset ();
	algoritms.F2_Ch.autoAVOM_canrun_flag:=FALSE;
	algoritms.F2_R.autoAVOM_canrun_flag:=FALSE;
END_IF
IF	(NOT algoritms.F2_Ch.autoAVOM_canrun_flag) AND (NOT algoritms.F2_R.autoAVOM_canrun_flag) AND pnsoff.start THEN
	Avom1Off.run ();
	Avom2Off.run ();
	Avom3Off.run ();
	Avom4Off.run ();
	algoritms.R_AutoAVOM.CanRun:=FALSE;
	algoritms.R_AutoAVOM.reset();
	algoritms.S_AutoAVOM.CanRun:=FALSE;
	algoritms.S_AutoAVOM.reset();
	algoritms.Auto_Avom_.CanRun:=FALSE;
	autoAVOMOff.run ();
END_IF
/////////////////////////////////////////
IF 	pnsOff.top AND Avom1Off.top AND Avom2Off.top AND Avom3Off.top AND Avom4Off.top AND autoAVOMOff.top  THEN //Если  отключен ПНС завершаем алгоритм
	end();
	timer5.run ();
END_IF
/////////////////////////////////////////
IF 	timer5.top THEN
	timer5.reset ();
	reset ();
END_IF

METHOD PUBLIC reset
VAR_INPUT
END_VAR
SUPER^.reset();
sbrosVibeg.reset();
statusSet.setBit(15,0);
flag1:=FALSE;
ystavki.Block_kr1_alg.setValue (0);
ystavki.Block_kr2_alg.setValue (0);
END_METHOD

METHOD PUBLIC run
VAR_INPUT
END_VAR
SUPER^.run();
algManager.setMode(nMode:=ModeGpa.MODE_AO);
statusSet.setBit(15,1);
IF	algmanager.reg_V THEN
	Start_AO_From.top:=TRUE;
END_IF
END_METHOD

END_FUNCTION_BLOCK

// K2/std12k5/ostanov/aoAlg
	{attribute 'symbol' := 'none'}
FUNCTION_BLOCK aoAlg EXTENDS StepBySteapAlgoritm
VAR_INPUT
END_VAR
VAR_OUTPUT
	{attribute 'symbol' := 'read'}
	sbrosVibeg:		Question(table:=ADR(ObjectTable)):=			(AnswerVariants:=Answers.ANS_YES);
END_VAR
VAR
	
	kran6Open:		ph_Kran (table:=ADR(phasesTable)):=				(phaseNumber:=0, Im:=Im.kran6, act:=DualStateImAction.on);
	
	kran4Close:		ph_Kran (table:=ADR(phasesTable)):=				(phaseNumber:=1, Im:=Im.kran4, act:=DualStateImAction.off);
	
	kran3bOpen:		ph_Kran (table:=ADR(phasesTable)):=				(phaseNumber:=2, Im:=Im.kran3b, act:=DualStateImAction.on);
	
	mvOff:			ph_Switch (table:=ADR(phasesTable)):=			(phaseNumber:=3, Im:=Im.mv, act:=DualStateImAction.off);
	
	kran1Close:		ph_Kran (table:=ADR(phasesTable)):=				(phaseNumber:=4, Im:=Im.kran1, act:=DualStateImAction.off);
	
	kran2Close:		ph_Kran (table:=ADR(phasesTable)):=				(phaseNumber:=5, Im:=Im.kran2, act:=DualStateImAction.off);
	
	kran3Close:		ph_Kran (table:=ADR(phasesTable)):=				(phaseNumber:=6, Im:=Im.kran3, act:=DualStateImAction.off);
	
	kran5Open:		ph_Kran (table:=ADR(phasesTable)):=				(phaseNumber:=7, Im:=Im.kran5, act:=DualStateImAction.on);
	
	autoPnsOff:		ph_algoritm (table:=ADR(phasesTable)):=			(phaseNumber:=8, Im:=algoritms.autoPns, act:=PhaseAlgoritmAction.reset, waitCompletion:=FALSE);
	
	pnsOn:			ph_Switch (table:=ADR(phasesTable)):=			(phaseNumber:=9, Im:=Im.pns, act:=DualStateImAction.on);
	
	Pg_VhodLessThen300:	CustomPhase (table:=ADR(phasesTable)):=		(phaseNumber:=10);
	
	Pg_VyhodLessThen300:CustomPhase (table:=ADR(phasesTable)):=		(phaseNumber:=11);
	
	nuOff:			ph_Switch (table:=ADR(phasesTable)):=			(phaseNumber:=12, Im:=Im.nu, act:=DualStateImAction.off);
	Auto_NU_Off:	CustomPhase (table:=ADR(phasesTable)):=		(phaseNumber:=13);
	{attribute 'symbol' := 'read'}
	timer600:		ph_Timer (table:=ADR(phasesTable)):=			(phaseNumber:=14, delay:=T#600S);
	
	pnsOff:			ph_Switch (table:=ADR(phasesTable)):=			(phaseNumber:=15, Im:=Im.pns, act:=DualStateImAction.off);
	
	Avom1Off:		ph_Switch (table:=ADR(phasesTable)):=			(phaseNumber:=16, Im:=Im.v1_Avom, act:=DualStateImAction.off);
	
	Avom2Off:		ph_Switch (table:=ADR(phasesTable)):=			(phaseNumber:=17, Im:=Im.v2_Avom, act:=DualStateImAction.off);
	
	Avom3Off:		ph_Switch (table:=ADR(phasesTable)):=			(phaseNumber:=18, Im:=Im.v3_Avom, act:=DualStateImAction.off);
	
	Avom4Off:		ph_Switch (table:=ADR(phasesTable)):=			(phaseNumber:=19, Im:=Im.v4_Avom, act:=DualStateImAction.off);
	
	autoAVOMOff:	ph_algoritm (table:=ADR(phasesTable)):=			(phaseNumber:=20, Im:=algoritms.Auto_Avom_, act:=PhaseAlgoritmAction.reset, waitCompletion:=FALSE);
	
	timer5:			ph_Timer (table:=ADR(phasesTable)):=			(phaseNumber:=21, delay:=T#5S);
	
	klapan1:		CustomPhase (table:=ADR(phasesTable)):=			(phaseNumber:=22);
	
	klapan2:		CustomPhase (table:=ADR(phasesTable)):=			(phaseNumber:=23);
	
